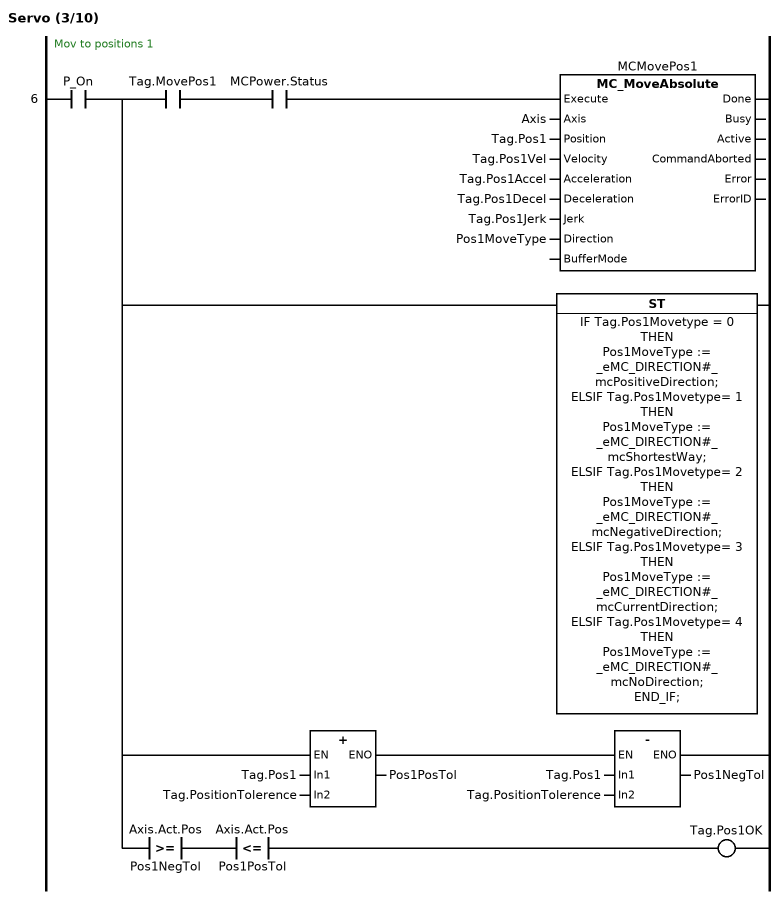
(* [picture p96: Servo, rungs 6-6] *)
(* Rung 6: Mov to positions 1 *)
MCMovePos1(Execute := P_On AND Tag.MovePos1 AND MCPower.Status, Axis := Axis, Position := Tag.Pos1, Velocity := Tag.Pos1Vel, Acceleration := Tag.Pos1Accel, Deceleration := Tag.Pos1Decel, Jerk := Tag.Pos1Jerk, Direction := Pos1MoveType);
IF P_On THEN
    IF Tag.Pos1Movetype = 0 THEN
    Pos1MoveType := _eMC_DIRECTION#_mcPositiveDirection;
    ELSIF Tag.Pos1Movetype= 1 THEN
    Pos1MoveType := _eMC_DIRECTION#_mcShortestWay;
    ELSIF Tag.Pos1Movetype= 2 THEN
    Pos1MoveType := _eMC_DIRECTION#_mcNegativeDirection;
    ELSIF Tag.Pos1Movetype= 3 THEN
    Pos1MoveType := _eMC_DIRECTION#_mcCurrentDirection;
    ELSIF Tag.Pos1Movetype= 4 THEN
    Pos1MoveType := _eMC_DIRECTION#_mcNoDirection;
    END_IF;
END_IF;
IF P_On THEN
    Pos1PosTol := Tag.Pos1 + Tag.PositionTolerence;
    Pos1NegTol := Tag.Pos1 - Tag.PositionTolerence;
END_IF;
Tag.Pos1OK := P_On AND (Axis.Act.Pos >= Pos1NegTol) AND (Axis.Act.Pos <= Pos1PosTol);

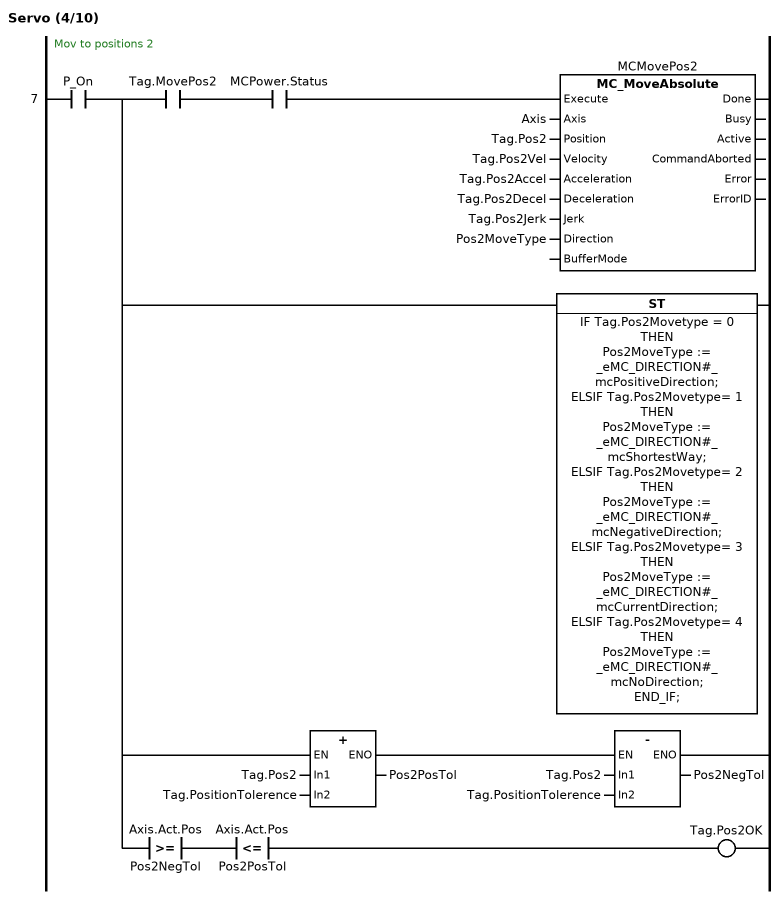
(* Rung 7: Mov to positions 2 *)
MCMovePos2(Execute := P_On AND Tag.MovePos2 AND MCPower.Status, Axis := Axis, Position := Tag.Pos2, Velocity := Tag.Pos2Vel, Acceleration := Tag.Pos2Accel, Deceleration := Tag.Pos2Decel, Jerk := Tag.Pos2Jerk, Direction := Pos2MoveType);
IF P_On THEN
    IF Tag.Pos2Movetype = 0 THEN
    Pos2MoveType := _eMC_DIRECTION#_mcPositiveDirection;
    ELSIF Tag.Pos2Movetype= 1 THEN
    Pos2MoveType := _eMC_DIRECTION#_mcShortestWay;
    ELSIF Tag.Pos2Movetype= 2 THEN
    Pos2MoveType := _eMC_DIRECTION#_mcNegativeDirection;
    ELSIF Tag.Pos2Movetype= 3 THEN
    Pos2MoveType := _eMC_DIRECTION#_mcCurrentDirection;
    ELSIF Tag.Pos2Movetype= 4 THEN
    Pos2MoveType := _eMC_DIRECTION#_mcNoDirection;
    END_IF;
END_IF;
IF P_On THEN
    Pos2PosTol := Tag.Pos2 + Tag.PositionTolerence;
    Pos2NegTol := Tag.Pos2 - Tag.PositionTolerence;
END_IF;
Tag.Pos2OK := P_On AND (Axis.Act.Pos >= Pos2NegTol) AND (Axis.Act.Pos <= Pos2PosTol);

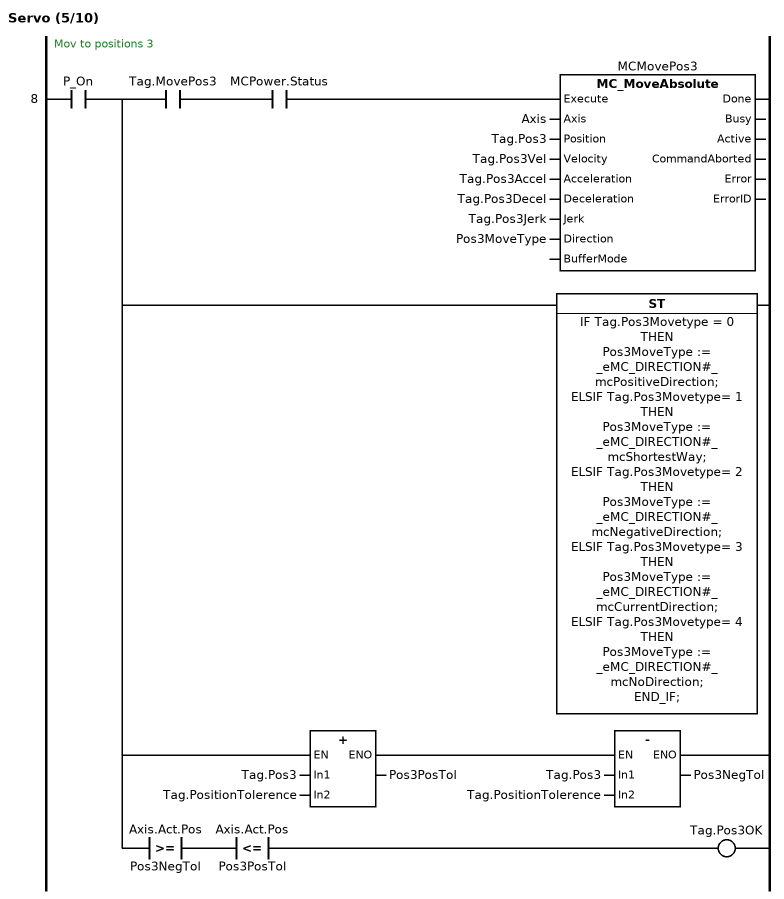
(* Rung 8: Mov to positions 3 *)
MCMovePos3(Execute := P_On AND Tag.MovePos3 AND MCPower.Status, Axis := Axis, Position := Tag.Pos3, Velocity := Tag.Pos3Vel, Acceleration := Tag.Pos3Accel, Deceleration := Tag.Pos3Decel, Jerk := Tag.Pos3Jerk, Direction := Pos3MoveType);
IF P_On THEN
    IF Tag.Pos3Movetype = 0 THEN
    Pos3MoveType := _eMC_DIRECTION#_mcPositiveDirection;
    ELSIF Tag.Pos3Movetype= 1 THEN
    Pos3MoveType := _eMC_DIRECTION#_mcShortestWay;
    ELSIF Tag.Pos3Movetype= 2 THEN
    Pos3MoveType := _eMC_DIRECTION#_mcNegativeDirection;
    ELSIF Tag.Pos3Movetype= 3 THEN
    Pos3MoveType := _eMC_DIRECTION#_mcCurrentDirection;
    ELSIF Tag.Pos3Movetype= 4 THEN
    Pos3MoveType := _eMC_DIRECTION#_mcNoDirection;
    END_IF;
END_IF;
IF P_On THEN
    Pos3PosTol := Tag.Pos3 + Tag.PositionTolerence;
    Pos3NegTol := Tag.Pos3 - Tag.PositionTolerence;
END_IF;
Tag.Pos3OK := P_On AND (Axis.Act.Pos >= Pos3NegTol) AND (Axis.Act.Pos <= Pos3PosTol);

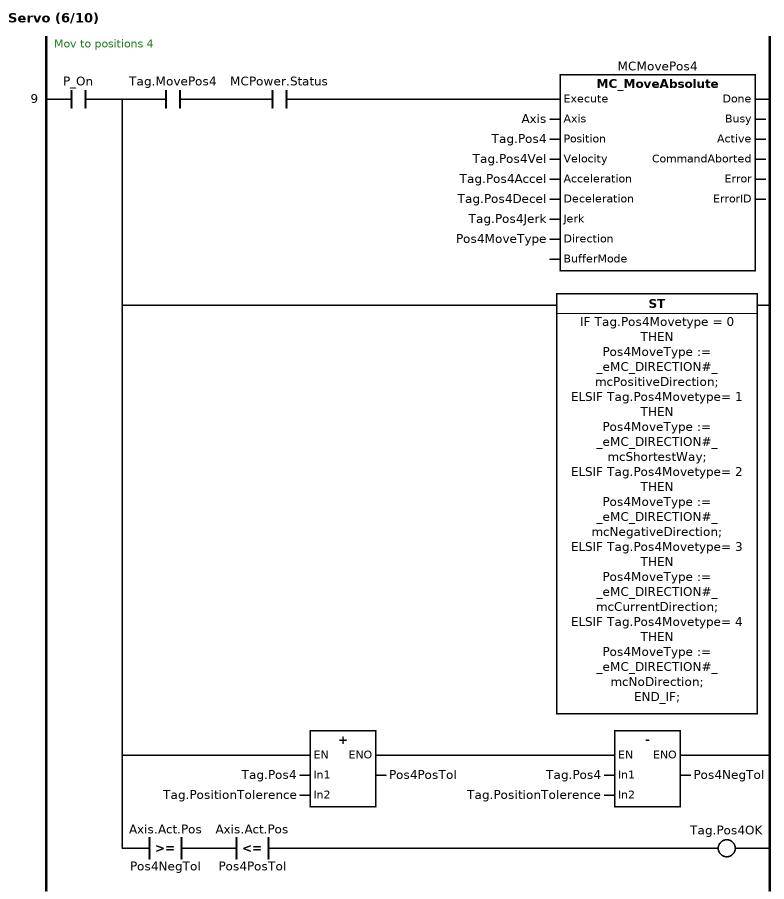
(* Rung 9: Mov to positions 4 *)
MCMovePos4(Execute := P_On AND Tag.MovePos4 AND MCPower.Status, Axis := Axis, Position := Tag.Pos4, Velocity := Tag.Pos4Vel, Acceleration := Tag.Pos4Accel, Deceleration := Tag.Pos4Decel, Jerk := Tag.Pos4Jerk, Direction := Pos4MoveType);
IF P_On THEN
    IF Tag.Pos4Movetype = 0 THEN
    Pos4MoveType := _eMC_DIRECTION#_mcPositiveDirection;
    ELSIF Tag.Pos4Movetype= 1 THEN
    Pos4MoveType := _eMC_DIRECTION#_mcShortestWay;
    ELSIF Tag.Pos4Movetype= 2 THEN
    Pos4MoveType := _eMC_DIRECTION#_mcNegativeDirection;
    ELSIF Tag.Pos4Movetype= 3 THEN
    Pos4MoveType := _eMC_DIRECTION#_mcCurrentDirection;
    ELSIF Tag.Pos4Movetype= 4 THEN
    Pos4MoveType := _eMC_DIRECTION#_mcNoDirection;
    END_IF;
END_IF;
IF P_On THEN
    Pos4PosTol := Tag.Pos4 + Tag.PositionTolerence;
    Pos4NegTol := Tag.Pos4 - Tag.PositionTolerence;
END_IF;
Tag.Pos4OK := P_On AND (Axis.Act.Pos >= Pos4NegTol) AND (Axis.Act.Pos <= Pos4PosTol);

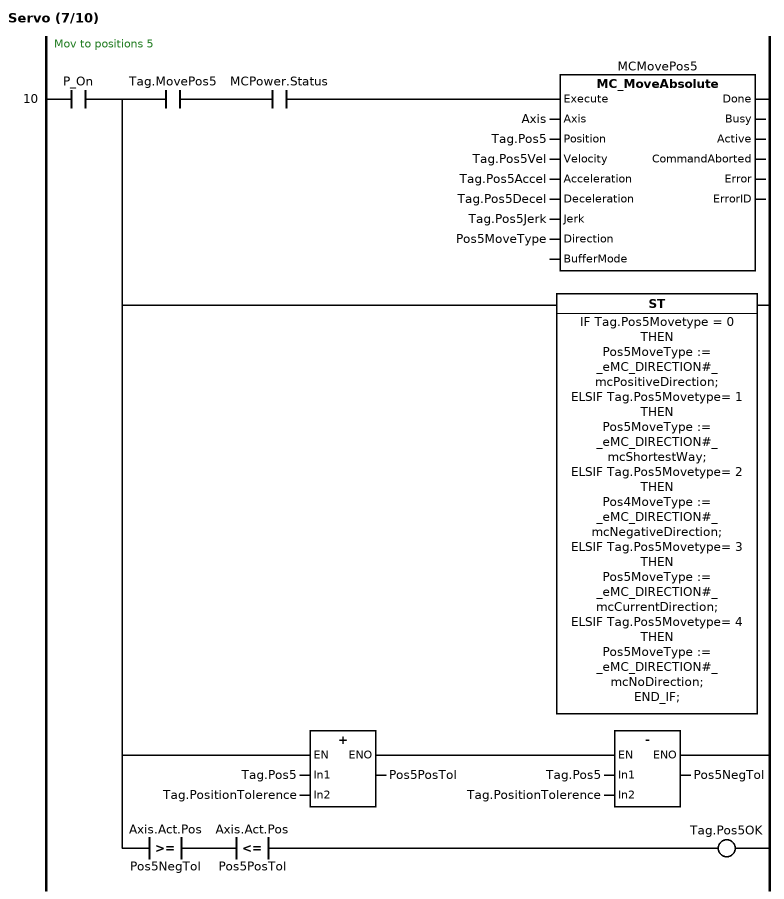
(* Rung 10: Mov to positions 5 *)
MCMovePos5(Execute := P_On AND Tag.MovePos5 AND MCPower.Status, Axis := Axis, Position := Tag.Pos5, Velocity := Tag.Pos5Vel, Acceleration := Tag.Pos5Accel, Deceleration := Tag.Pos5Decel, Jerk := Tag.Pos5Jerk, Direction := Pos5MoveType);
IF P_On THEN
    IF Tag.Pos5Movetype = 0 THEN
    Pos5MoveType := _eMC_DIRECTION#_mcPositiveDirection;
    ELSIF Tag.Pos5Movetype= 1 THEN
    Pos5MoveType := _eMC_DIRECTION#_mcShortestWay;
    ELSIF Tag.Pos5Movetype= 2 THEN
    Pos4MoveType := _eMC_DIRECTION#_mcNegativeDirection;
    ELSIF Tag.Pos5Movetype= 3 THEN
    Pos5MoveType := _eMC_DIRECTION#_mcCurrentDirection;
    ELSIF Tag.Pos5Movetype= 4 THEN
    Pos5MoveType := _eMC_DIRECTION#_mcNoDirection;
    END_IF;
END_IF;
IF P_On THEN
    Pos5PosTol := Tag.Pos5 + Tag.PositionTolerence;
    Pos5NegTol := Tag.Pos5 - Tag.PositionTolerence;
END_IF;
Tag.Pos5OK := P_On AND (Axis.Act.Pos >= Pos5NegTol) AND (Axis.Act.Pos <= Pos5PosTol);

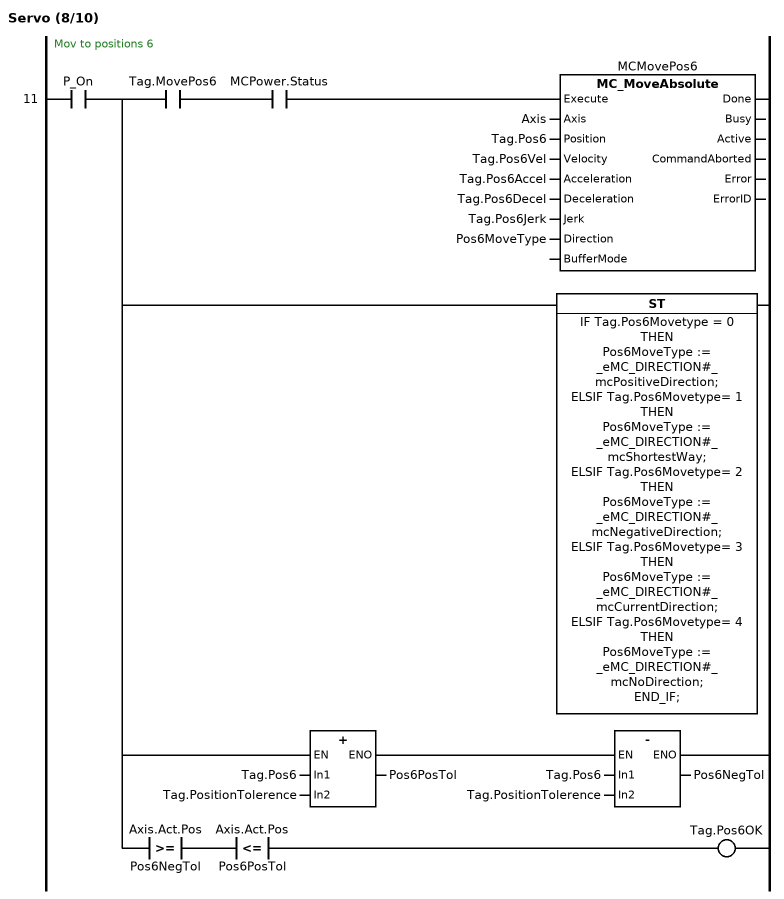
(* Rung 11: Mov to positions 6 *)
MCMovePos6(Execute := P_On AND Tag.MovePos6 AND MCPower.Status, Axis := Axis, Position := Tag.Pos6, Velocity := Tag.Pos6Vel, Acceleration := Tag.Pos6Accel, Deceleration := Tag.Pos6Decel, Jerk := Tag.Pos6Jerk, Direction := Pos6MoveType);
IF P_On THEN
    IF Tag.Pos6Movetype = 0 THEN
    Pos6MoveType := _eMC_DIRECTION#_mcPositiveDirection;
    ELSIF Tag.Pos6Movetype= 1 THEN
    Pos6MoveType := _eMC_DIRECTION#_mcShortestWay;
    ELSIF Tag.Pos6Movetype= 2 THEN
    Pos6MoveType := _eMC_DIRECTION#_mcNegativeDirection;
    ELSIF Tag.Pos6Movetype= 3 THEN
    Pos6MoveType := _eMC_DIRECTION#_mcCurrentDirection;
    ELSIF Tag.Pos6Movetype= 4 THEN
    Pos6MoveType := _eMC_DIRECTION#_mcNoDirection;
    END_IF;
END_IF;
IF P_On THEN
    Pos6PosTol := Tag.Pos6 + Tag.PositionTolerence;
    Pos6NegTol := Tag.Pos6 - Tag.PositionTolerence;
END_IF;
Tag.Pos6OK := P_On AND (Axis.Act.Pos >= Pos6NegTol) AND (Axis.Act.Pos <= Pos6PosTol);

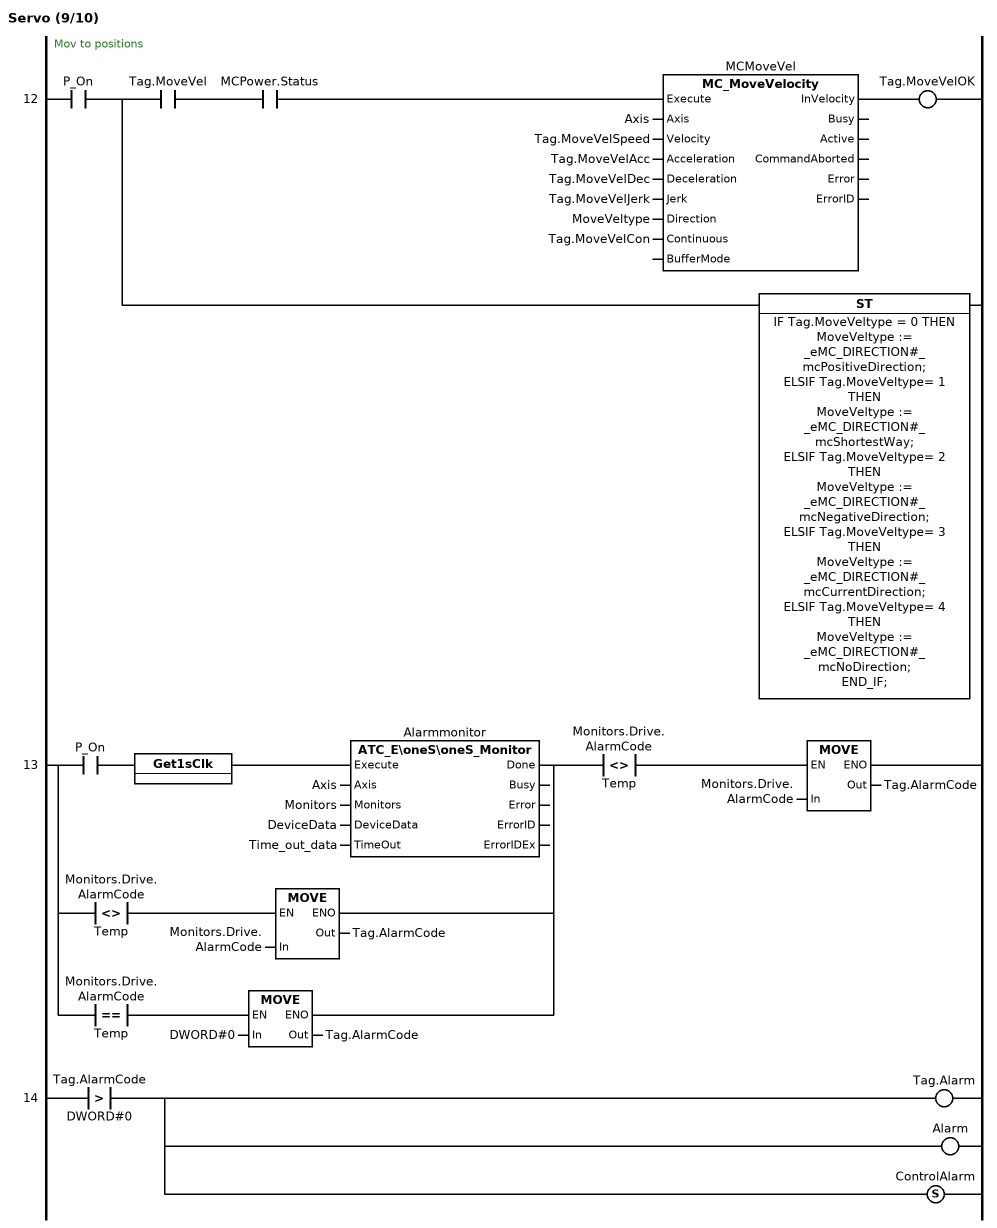
(* Rung 12: Mov to positions *)
MCMoveVel(Execute := P_On AND Tag.MoveVel AND MCPower.Status, Axis := Axis, Velocity := Tag.MoveVelSpeed, Acceleration := Tag.MoveVelAcc, Deceleration := Tag.MoveVelDec, Jerk := Tag.MoveVelJerk, Direction := MoveVeltype, Continuous := Tag.MoveVelCon);
Tag.MoveVelOK := MCMoveVel.InVelocity;
IF P_On THEN
    IF Tag.MoveVeltype = 0 THEN
    MoveVeltype := _eMC_DIRECTION#_mcPositiveDirection;
    ELSIF Tag.MoveVeltype= 1 THEN
    MoveVeltype := _eMC_DIRECTION#_mcShortestWay;
    ELSIF Tag.MoveVeltype= 2 THEN
    MoveVeltype := _eMC_DIRECTION#_mcNegativeDirection;
    ELSIF Tag.MoveVeltype= 3 THEN
    MoveVeltype := _eMC_DIRECTION#_mcCurrentDirection;
    ELSIF Tag.MoveVeltype= 4 THEN
    MoveVeltype := _eMC_DIRECTION#_mcNoDirection;
    END_IF;
END_IF;
(* Rung 13 *)
Alarmmonitor(Execute := P_On AND Get1sClk(), Axis := Axis, Monitors := Monitors, DeviceData := DeviceData, TimeOut := Time_out_data);
IF Monitors.Drive.AlarmCode <> Temp THEN Tag.AlarmCode := Monitors.Drive.AlarmCode; END_IF;
IF Monitors.Drive.AlarmCode = Temp THEN Tag.AlarmCode := DWORD#0; END_IF;
IF (Alarmmonitor.Done OR (Monitors.Drive.AlarmCode <> Temp) OR (Monitors.Drive.AlarmCode = Temp)) AND (Monitors.Drive.AlarmCode <> Temp) THEN
    Tag.AlarmCode := Monitors.Drive.AlarmCode;
END_IF;
(* Rung 14 *)
_p1 := Tag.AlarmCode > DWORD#0;
Tag.Alarm := _p1;
Alarm := _p1;
IF _p1 THEN ControlAlarm := TRUE; END_IF;

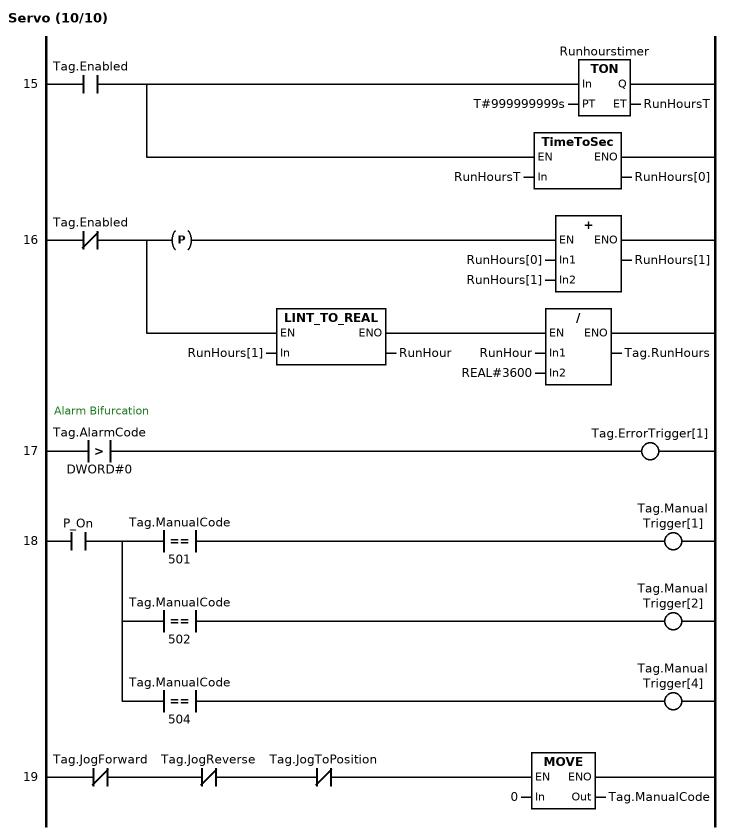
(* Rung 15 *)
Runhourstimer(In := Tag.Enabled, PT := T#999999999s, ET => RunHoursT);
IF Tag.Enabled THEN RunHours[0] := TimeToSec(In := RunHoursT); END_IF;
(* Rung 16 *)
_e2(CLK := NOT Tag.Enabled);
IF _e2.Q THEN RunHours[1] := RunHours[0] + RunHours[1]; END_IF;
IF NOT Tag.Enabled THEN
    RunHour := LINT_TO_REAL(In := RunHours[1]);
    Tag.RunHours := RunHour / REAL#3600;
END_IF;
(* Rung 17: Alarm Bifurcation *)
Tag.ErrorTrigger[1] := Tag.AlarmCode > DWORD#0;
(* Rung 18 *)
Tag.ManualTrigger[1] := P_On AND (Tag.ManualCode = 501);
Tag.ManualTrigger[2] := P_On AND (Tag.ManualCode = 502);
Tag.ManualTrigger[4] := P_On AND (Tag.ManualCode = 504);
(* Rung 19 *)
IF NOT Tag.JogForward AND NOT Tag.JogReverse AND NOT Tag.JogToPosition THEN Tag.ManualCode := 0; END_IF;
END_FUNCTION_BLOCK

FUNCTION_BLOCK MiscIN
VAR
    Powerup : BOOL;
    IN : BOOL;
    DebounceON : TON;
    Debounceoff : TON;
    In_Fault_Timer : TON;
    Timecal1 : LREAL;
    Timecal2 : LINT;
    DebounceONtime : TIME;
    Timecal3 : LINT;
    Timecal4 : LREAL;
    AccumulatedON : TIME;
    Timecal5 : LREAL;
    Timecal6 : LINT;
    DebounceOFFtime : TIME;
    Timecal7 : LINT;
    Timecal8 : LREAL;
    AccumulatedOFF : TIME;
    Timecal9 : LREAL;
    Timecal10 : LINT;
    Input_Fault_Time : TIME;
    Timecal11 : LINT;
    Timecal12 : LREAL;
    Input_Fault_Time_Acc : TIME;
END_VAR
VAR_OUTPUT
    EnableOut : BOOL;
END_VAR
VAR_INPUT
    input : BOOL;
    Accnowledge : BOOL;
END_VAR
VAR_IN_OUT
    tag : MiscInD;
END_VAR
VAR_OUTPUT
    Alarm : BOOL;
END_VAR
VAR_IN_OUT
    ControlAlarm : BOOL;
END_VAR
VAR
    _p1 : BOOL;
    _p2 : BOOL;
    _p3 : BOOL;
    _p4 : BOOL;
    _p5 : BOOL;
END_VAR
(* ladder, written here as Structured Text *)

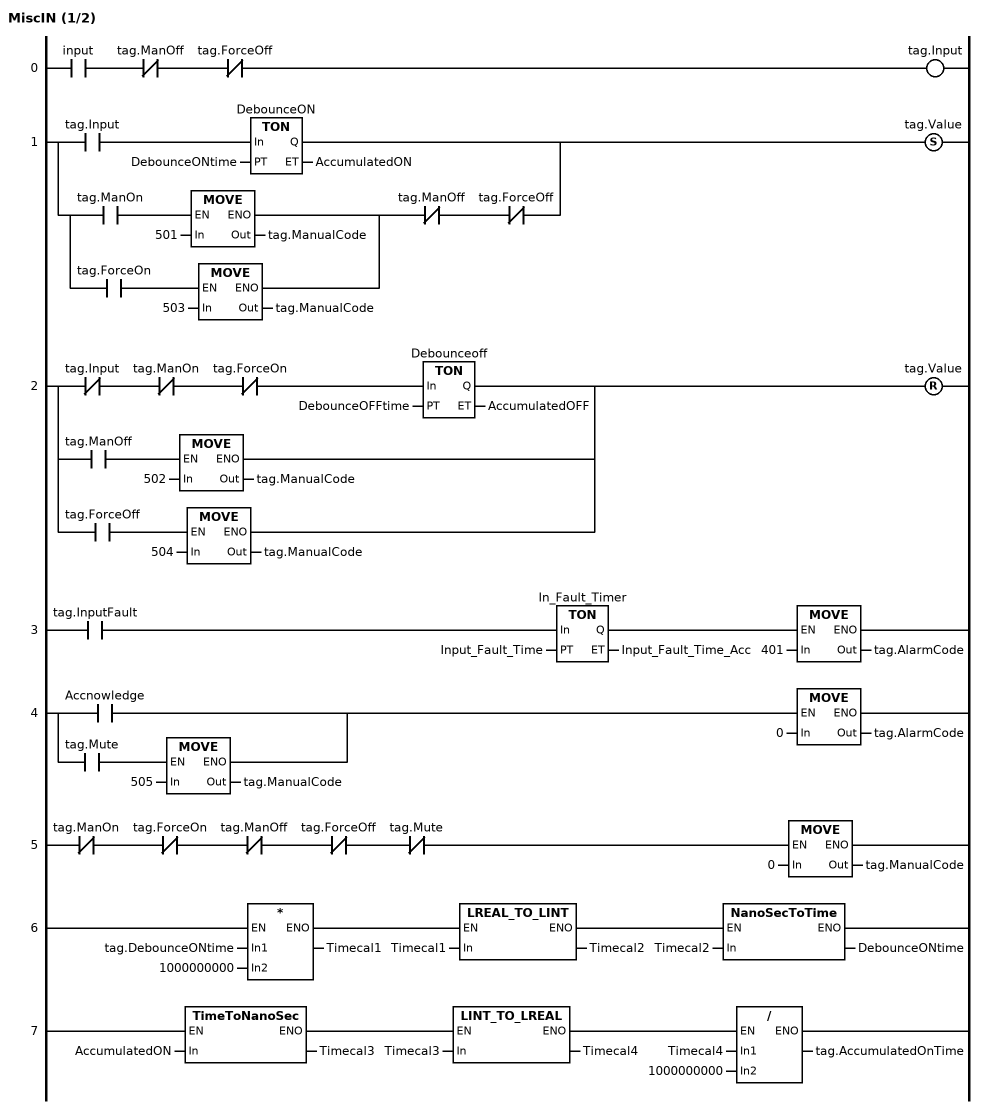
(* Rung 0 *)
tag.Input := input AND NOT tag.ManOff AND NOT tag.ForceOff;
(* Rung 1 *)
DebounceON(In := tag.Input, PT := DebounceONtime, ET => AccumulatedON);
_p1 := tag.ManOn;
IF _p1 THEN tag.ManualCode := 501; END_IF;
_p2 := tag.ForceOn;
IF _p2 THEN tag.ManualCode := 503; END_IF;
IF DebounceON.Q OR ((_p1 OR _p2) AND NOT tag.ManOff AND NOT tag.ForceOff) THEN tag.Value := TRUE; END_IF;
(* Rung 2 *)
Debounceoff(In := NOT tag.Input AND NOT tag.ManOn AND NOT tag.ForceOn, PT := DebounceOFFtime, ET => AccumulatedOFF);
_p3 := tag.ManOff;
IF _p3 THEN tag.ManualCode := 502; END_IF;
_p4 := tag.ForceOff;
IF _p4 THEN tag.ManualCode := 504; END_IF;
IF Debounceoff.Q OR _p3 OR _p4 THEN tag.Value := FALSE; END_IF;
(* Rung 3 *)
In_Fault_Timer(In := tag.InputFault, PT := Input_Fault_Time, ET => Input_Fault_Time_Acc);
IF In_Fault_Timer.Q THEN tag.AlarmCode := 401; END_IF;
(* Rung 4 *)
_p5 := tag.Mute;
IF _p5 THEN tag.ManualCode := 505; END_IF;
IF Accnowledge OR _p5 THEN tag.AlarmCode := 0; END_IF;
(* Rung 5 *)
IF NOT tag.ManOn AND NOT tag.ForceOn AND NOT tag.ManOff AND NOT tag.ForceOff AND NOT tag.Mute THEN
    tag.ManualCode := 0;
END_IF;
(* Rung 6 *)
Timecal1 := tag.DebounceONtime * 1000000000;
Timecal2 := LREAL_TO_LINT(In := Timecal1);
DebounceONtime := NanoSecToTime(In := Timecal2);
(* Rung 7 *)
Timecal3 := TimeToNanoSec(In := AccumulatedON);
Timecal4 := LINT_TO_LREAL(In := Timecal3);
tag.AccumulatedOnTime := Timecal4 / 1000000000;

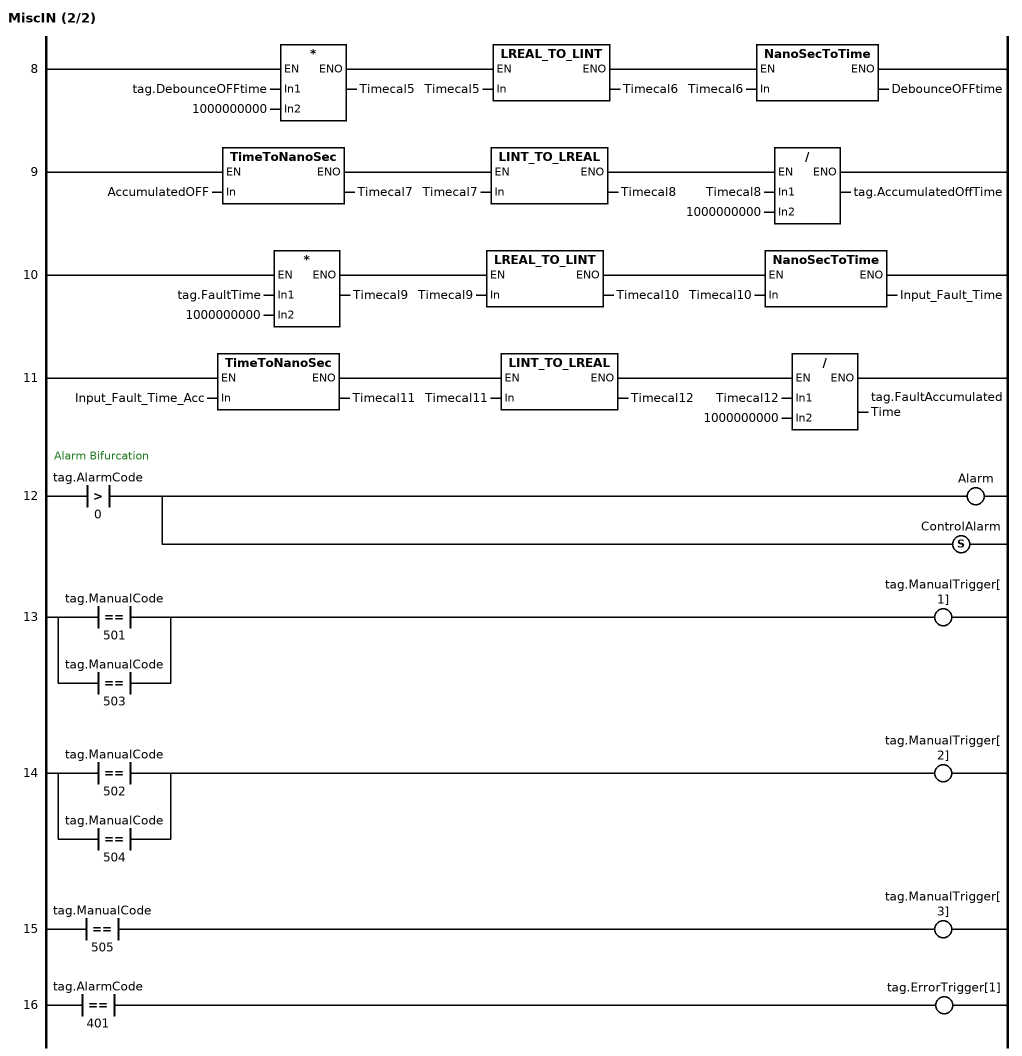
(* Rung 8 *)
Timecal5 := tag.DebounceOFFtime * 1000000000;
Timecal6 := LREAL_TO_LINT(In := Timecal5);
DebounceOFFtime := NanoSecToTime(In := Timecal6);
(* Rung 9 *)
Timecal7 := TimeToNanoSec(In := AccumulatedOFF);
Timecal8 := LINT_TO_LREAL(In := Timecal7);
tag.AccumulatedOffTime := Timecal8 / 1000000000;
(* Rung 10 *)
Timecal9 := tag.FaultTime * 1000000000;
Timecal10 := LREAL_TO_LINT(In := Timecal9);
Input_Fault_Time := NanoSecToTime(In := Timecal10);
(* Rung 11 *)
Timecal11 := TimeToNanoSec(In := Input_Fault_Time_Acc);
Timecal12 := LINT_TO_LREAL(In := Timecal11);
tag.FaultAccumulatedTime := Timecal12 / 1000000000;
(* Rung 12: Alarm Bifurcation *)
Alarm := tag.AlarmCode > 0;
IF tag.AlarmCode > 0 THEN ControlAlarm := TRUE; END_IF;
(* Rung 13 *)
tag.ManualTrigger[1] := (tag.ManualCode = 501) OR (tag.ManualCode = 503);
(* Rung 14 *)
tag.ManualTrigger[2] := (tag.ManualCode = 502) OR (tag.ManualCode = 504);
(* Rung 15 *)
tag.ManualTrigger[3] := tag.ManualCode = 505;
(* Rung 16 *)
tag.ErrorTrigger[1] := tag.AlarmCode = 401;
END_FUNCTION_BLOCK

FUNCTION_BLOCK Motor
VAR
    Forward : BOOL;
    Reverse : BOOL;
    FeedBackOffTimer : TON;
END_VAR
VAR RETAIN
    Faulttime : TIME;
END_VAR
VAR
    MotorFault : BOOL;
    FeedBackOnTimer : TON;
    Faulttime1Acc : TIME;
    MotorFaultRev : BOOL;
    Timecal7 : LREAL;
    Timecal8 : LINT;
    Timecal9 : LINT;
    Timecal10 : LREAL;
    FaulttimeAcc : TIME;
    RunHoursT : TIME;
    RunHours : ARRAY[0..1] OF LINT;
    RunHour : REAL;
    RunHoursTimer : TON;
    MotorFaultoff : BOOL;
    FeedBackOffTimer1 : TON;
END_VAR
VAR_INPUT
    Enable : BOOL;
END_VAR
VAR_OUTPUT
    Enableout : BOOL;
    OutputForward : BOOL;
    OutputReverse : BOOL;
END_VAR
VAR_INPUT
    RunFeedBack : BOOL;
END_VAR
VAR_IN_OUT
    Tag : MotorD;
END_VAR
VAR_OUTPUT
    Alarm : BOOL;
END_VAR
VAR_IN_OUT
    ControlCom : System;
END_VAR
VAR
    _e1 : R_TRIG;
    _e2 : R_TRIG;
    _p3 : BOOL;
    _e4 : R_TRIG;
    _e5 : R_TRIG;
    _p6 : BOOL;
    _p7 : BOOL;
    _p8 : BOOL;
    _p9 : BOOL;
    _e10 : R_TRIG;
    _e11 : R_TRIG;
    _p12 : BOOL;
END_VAR
(* ladder, written here as Structured Text *)

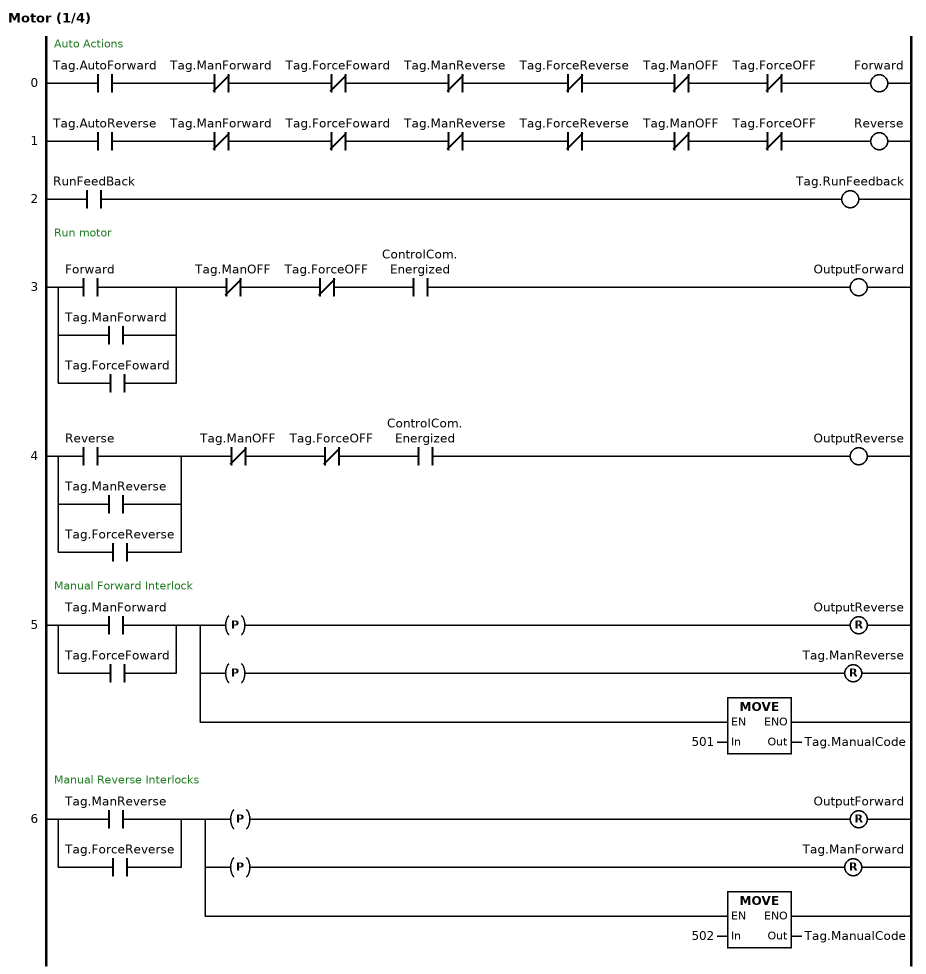
(* Rung 0: Auto Actions *)
Forward := Tag.AutoForward AND NOT Tag.ManForward AND NOT Tag.ForceFoward AND NOT Tag.ManReverse AND NOT Tag.ForceReverse AND NOT Tag.ManOFF AND NOT Tag.ForceOFF;
(* Rung 1 *)
Reverse := Tag.AutoReverse AND NOT Tag.ManForward AND NOT Tag.ForceFoward AND NOT Tag.ManReverse AND NOT Tag.ForceReverse AND NOT Tag.ManOFF AND NOT Tag.ForceOFF;
(* Rung 2 *)
Tag.RunFeedback := RunFeedBack;
(* Rung 3: Run motor *)
OutputForward := (Forward OR Tag.ManForward OR Tag.ForceFoward) AND NOT Tag.ManOFF AND NOT Tag.ForceOFF AND ControlCom.Energized;
(* Rung 4 *)
OutputReverse := (Reverse OR Tag.ManReverse OR Tag.ForceReverse) AND NOT Tag.ManOFF AND NOT Tag.ForceOFF AND ControlCom.Energized;
(* Rung 5: Manual Forward Interlock *)
_e1(CLK := Tag.ManForward OR Tag.ForceFoward);
IF _e1.Q THEN OutputReverse := FALSE; END_IF;
_e2(CLK := Tag.ManForward OR Tag.ForceFoward);
_p3 := Tag.ManForward OR Tag.ForceFoward;
IF _e2.Q THEN Tag.ManReverse := FALSE; END_IF;
IF _p3 THEN Tag.ManualCode := 501; END_IF;
(* Rung 6: Manual Reverse Interlocks *)
_e4(CLK := Tag.ManReverse OR Tag.ForceReverse);
IF _e4.Q THEN OutputForward := FALSE; END_IF;
_e5(CLK := Tag.ManReverse OR Tag.ForceReverse);
_p6 := Tag.ManReverse OR Tag.ForceReverse;
IF _e5.Q THEN Tag.ManForward := FALSE; END_IF;
IF _p6 THEN Tag.ManualCode := 502; END_IF;

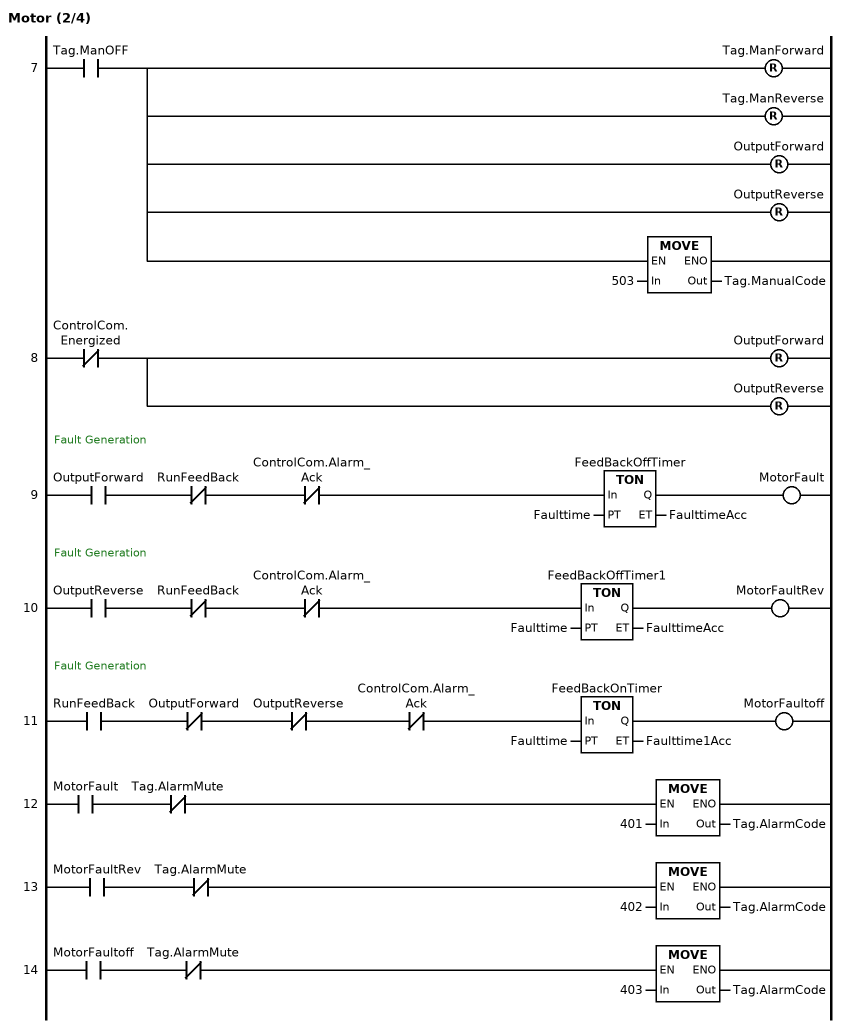
(* Rung 7 *)
_p7 := Tag.ManOFF;
IF _p7 THEN
    Tag.ManForward := FALSE;
    Tag.ManReverse := FALSE;
    OutputForward := FALSE;
    OutputReverse := FALSE;
    Tag.ManualCode := 503;
END_IF;
(* Rung 8 *)
IF NOT ControlCom.Energized THEN
    OutputForward := FALSE;
    OutputReverse := FALSE;
END_IF;
(* Rung 9: Fault Generation *)
FeedBackOffTimer(In := OutputForward AND NOT RunFeedBack AND NOT ControlCom.Alarm_Ack, PT := Faulttime, ET => FaulttimeAcc);
MotorFault := FeedBackOffTimer.Q;
(* Rung 10: Fault Generation *)
FeedBackOffTimer1(In := OutputReverse AND NOT RunFeedBack AND NOT ControlCom.Alarm_Ack, PT := Faulttime, ET => FaulttimeAcc);
MotorFaultRev := FeedBackOffTimer1.Q;
(* Rung 11: Fault Generation *)
FeedBackOnTimer(In := RunFeedBack AND NOT OutputForward AND NOT OutputReverse AND NOT ControlCom.Alarm_Ack, PT := Faulttime, ET => Faulttime1Acc);
MotorFaultoff := FeedBackOnTimer.Q;
(* Rung 12 *)
IF MotorFault AND NOT Tag.AlarmMute THEN Tag.AlarmCode := 401; END_IF;
(* Rung 13 *)
IF MotorFaultRev AND NOT Tag.AlarmMute THEN Tag.AlarmCode := 402; END_IF;
(* Rung 14 *)
IF MotorFaultoff AND NOT Tag.AlarmMute THEN Tag.AlarmCode := 403; END_IF;

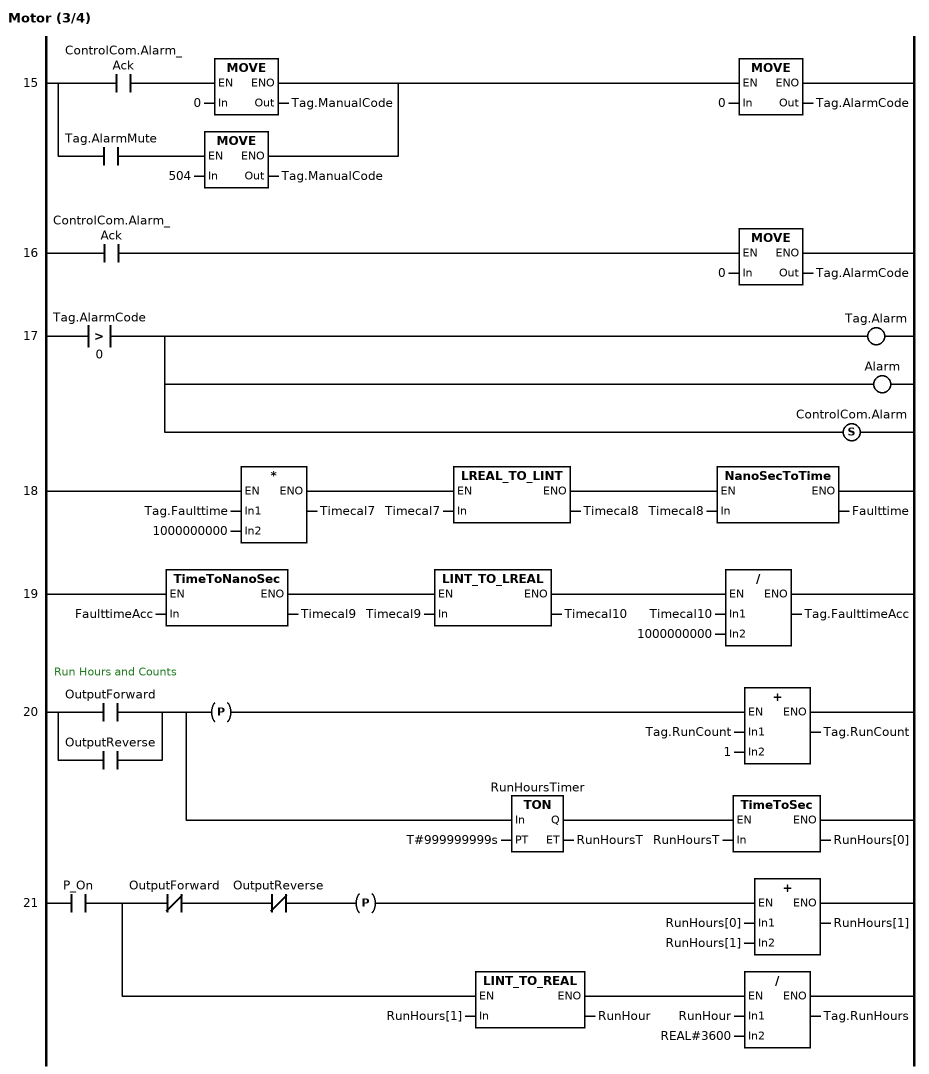
(* Rung 15 *)
IF ControlCom.Alarm_Ack THEN Tag.ManualCode := 0; END_IF;
_p8 := Tag.AlarmMute;
IF _p8 THEN Tag.ManualCode := 504; END_IF;
IF ControlCom.Alarm_Ack OR _p8 THEN Tag.AlarmCode := 0; END_IF;
(* Rung 16 *)
IF ControlCom.Alarm_Ack THEN Tag.AlarmCode := 0; END_IF;
(* Rung 17 *)
_p9 := Tag.AlarmCode > 0;
Tag.Alarm := _p9;
Alarm := _p9;
IF _p9 THEN ControlCom.Alarm := TRUE; END_IF;
(* Rung 18 *)
Timecal7 := Tag.Faulttime * 1000000000;
Timecal8 := LREAL_TO_LINT(In := Timecal7);
Faulttime := NanoSecToTime(In := Timecal8);
(* Rung 19 *)
Timecal9 := TimeToNanoSec(In := FaulttimeAcc);
Timecal10 := LINT_TO_LREAL(In := Timecal9);
Tag.FaulttimeAcc := Timecal10 / 1000000000;
(* Rung 20: Run Hours and Counts *)
_e10(CLK := OutputForward OR OutputReverse);
IF _e10.Q THEN Tag.RunCount := Tag.RunCount + 1; END_IF;
RunHoursTimer(In := OutputForward OR OutputReverse, PT := T#999999999s, ET => RunHoursT);
IF RunHoursTimer.Q THEN RunHours[0] := TimeToSec(In := RunHoursT); END_IF;
(* Rung 21 *)
_e11(CLK := P_On AND NOT OutputForward AND NOT OutputReverse);
IF _e11.Q THEN RunHours[1] := RunHours[0] + RunHours[1]; END_IF;
IF P_On THEN
    RunHour := LINT_TO_REAL(In := RunHours[1]);
    Tag.RunHours := RunHour / REAL#3600;
END_IF;

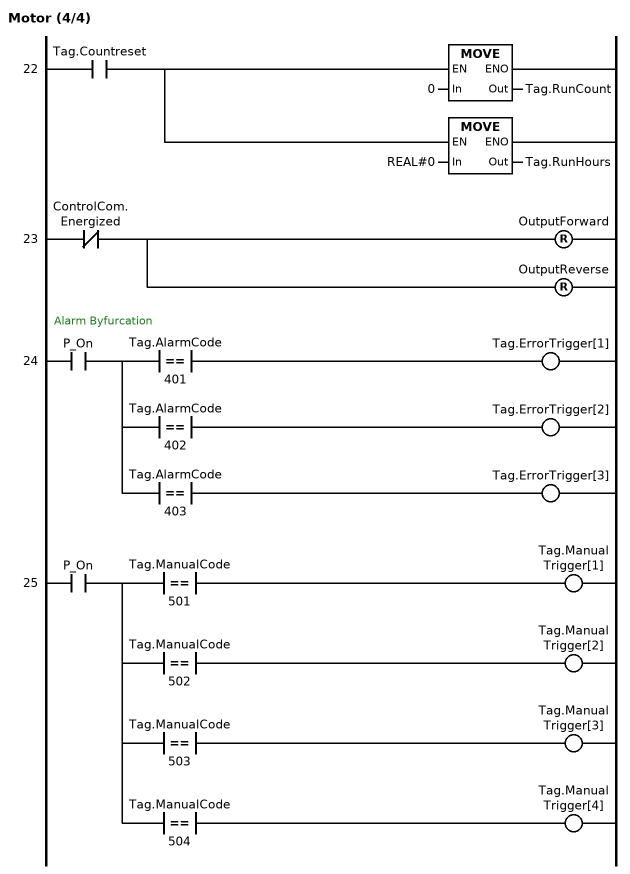
(* Rung 22 *)
_p12 := Tag.Countreset;
IF _p12 THEN
    Tag.RunCount := 0;
    Tag.RunHours := REAL#0;
END_IF;
(* Rung 23 *)
IF NOT ControlCom.Energized THEN
    OutputForward := FALSE;
    OutputReverse := FALSE;
END_IF;
(* Rung 24: Alarm Byfurcation *)
Tag.ErrorTrigger[1] := P_On AND (Tag.AlarmCode = 401);
Tag.ErrorTrigger[2] := P_On AND (Tag.AlarmCode = 402);
Tag.ErrorTrigger[3] := P_On AND (Tag.AlarmCode = 403);
(* Rung 25 *)
Tag.ManualTrigger[1] := P_On AND (Tag.ManualCode = 501);
Tag.ManualTrigger[2] := P_On AND (Tag.ManualCode = 502);
Tag.ManualTrigger[3] := P_On AND (Tag.ManualCode = 503);
Tag.ManualTrigger[4] := P_On AND (Tag.ManualCode = 504);
END_FUNCTION_BLOCK

FUNCTION_BLOCK MotorVSD
VAR
    Forward : BOOL;
    Reverse : BOOL;
    FeedBackOffTimer : TON;
END_VAR
VAR RETAIN
    Faulttime : TIME;
END_VAR
VAR
    MotorFault : BOOL;
    FeedBackOnTimer : TON;
    Faulttime1Acc : TIME;
    MotorFaultRev : BOOL;
    Timecal7 : LREAL;
    Timecal8 : LINT;
    Timecal9 : LINT;
    Timecal10 : LREAL;
    FaulttimeAcc : TIME;
    OutputForward : BOOL;
    OutputReverse : BOOL;
    MotorFaultFor : BOOL;
    FeedBackOffTimerFor : TON;
    FeedBackOnTimerRev : TON;
    Faulttime2Acc : TIME;
    RunHoursTimer : TON;
    RunHoursT : TIME;
    RunHours : ARRAY[0..1] OF LINT;
    RunHour : REAL;
END_VAR
VAR_INPUT
    Enable : BOOL;
END_VAR
VAR_OUTPUT
    Enableout : BOOL;
END_VAR
VAR_IN_OUT
    Tag : MotorVSDD;
END_VAR
VAR_OUTPUT
    DirectionOut : WORD;
    SpeedOut : UINT;
END_VAR
VAR_INPUT
    RunFeedBack : WORD;
END_VAR
VAR_OUTPUT
    Alarm : BOOL;
END_VAR
VAR_IN_OUT
    ControlCom : System;
END_VAR
VAR_EXTERNAL
    Zcomm : ARRAY[0..31] OF BOOL;
END_VAR
VAR
    _p1 : BOOL;
    _e2 : R_TRIG;
    _e3 : R_TRIG;
    _p4 : BOOL;
    _e5 : R_TRIG;
    _e6 : R_TRIG;
    _p7 : BOOL;
    _p8 : BOOL;
    _p9 : BOOL;
    _e10 : R_TRIG;
    _e11 : R_TRIG;
    _p12 : BOOL;
END_VAR
(* ladder, written here as Structured Text *)

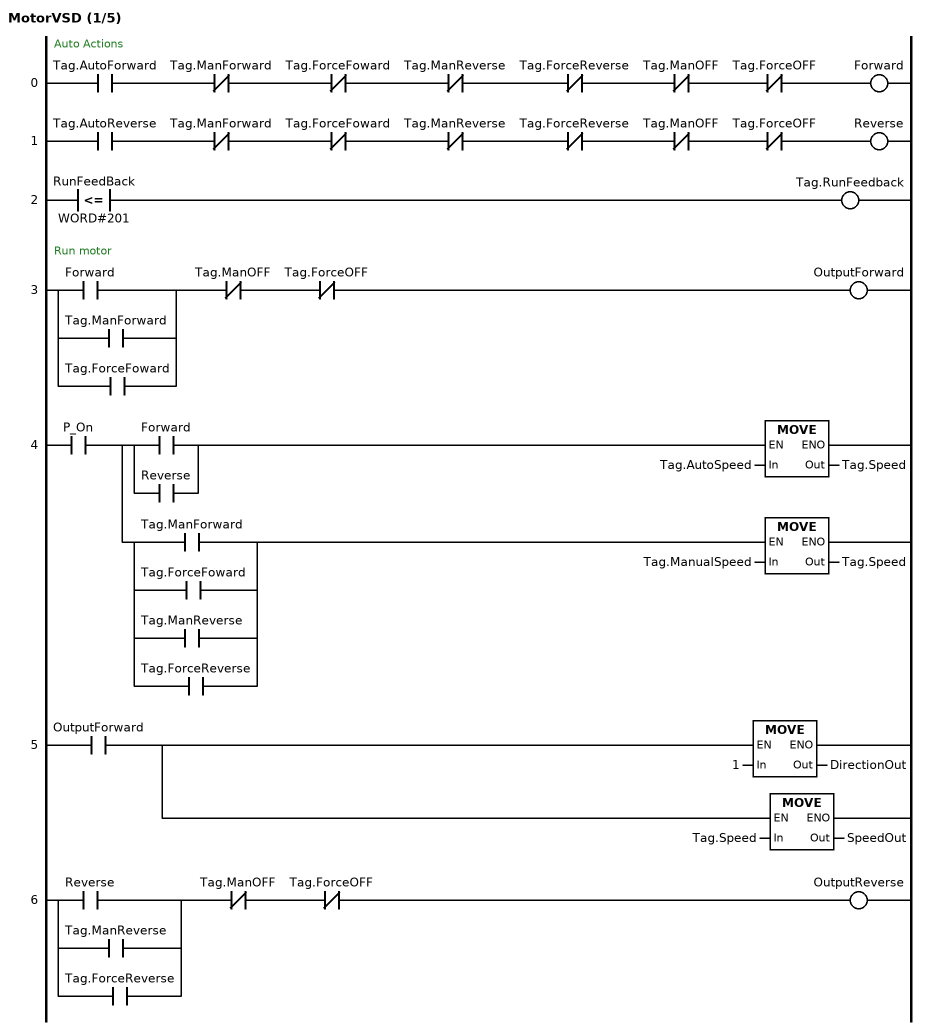
(* Rung 0: Auto Actions *)
Forward := Tag.AutoForward AND NOT Tag.ManForward AND NOT Tag.ForceFoward AND NOT Tag.ManReverse AND NOT Tag.ForceReverse AND NOT Tag.ManOFF AND NOT Tag.ForceOFF;
(* Rung 1 *)
Reverse := Tag.AutoReverse AND NOT Tag.ManForward AND NOT Tag.ForceFoward AND NOT Tag.ManReverse AND NOT Tag.ForceReverse AND NOT Tag.ManOFF AND NOT Tag.ForceOFF;
(* Rung 2 *)
Tag.RunFeedback := RunFeedBack <= WORD#201;
(* Rung 3: Run motor *)
OutputForward := (Forward OR Tag.ManForward OR Tag.ForceFoward) AND NOT Tag.ManOFF AND NOT Tag.ForceOFF;
(* Rung 4 *)
IF P_On AND (Forward OR Reverse) THEN Tag.Speed := Tag.AutoSpeed; END_IF;
IF P_On AND (Tag.ManForward OR Tag.ForceFoward OR Tag.ManReverse OR Tag.ForceReverse) THEN
    Tag.Speed := Tag.ManualSpeed;
END_IF;
(* Rung 5 *)
IF OutputForward THEN
    DirectionOut := 1;
    SpeedOut := Tag.Speed;
END_IF;
(* Rung 6 *)
OutputReverse := (Reverse OR Tag.ManReverse OR Tag.ForceReverse) AND NOT Tag.ManOFF AND NOT Tag.ForceOFF;

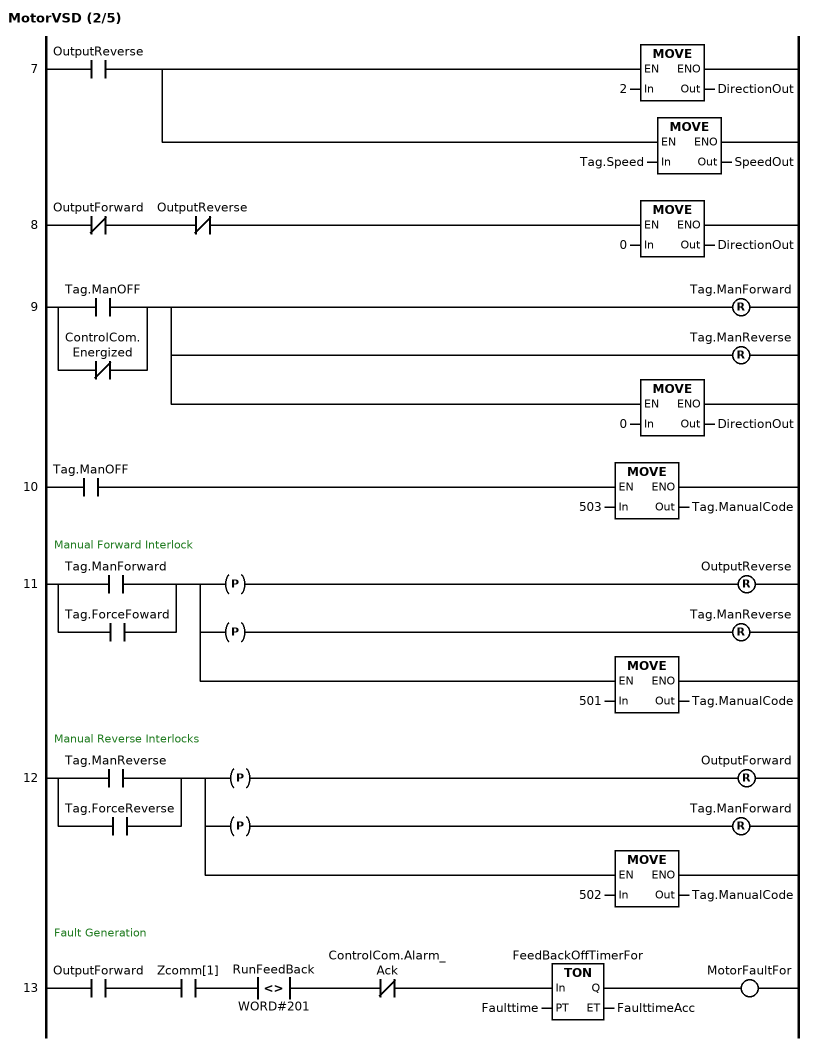
(* Rung 7 *)
IF OutputReverse THEN
    DirectionOut := 2;
    SpeedOut := Tag.Speed;
END_IF;
(* Rung 8 *)
IF NOT OutputForward AND NOT OutputReverse THEN DirectionOut := 0; END_IF;
(* Rung 9 *)
_p1 := Tag.ManOFF OR NOT ControlCom.Energized;
IF _p1 THEN
    Tag.ManForward := FALSE;
    Tag.ManReverse := FALSE;
    DirectionOut := 0;
END_IF;
(* Rung 10 *)
IF Tag.ManOFF THEN Tag.ManualCode := 503; END_IF;
(* Rung 11: Manual Forward Interlock *)
_e2(CLK := Tag.ManForward OR Tag.ForceFoward);
IF _e2.Q THEN OutputReverse := FALSE; END_IF;
_e3(CLK := Tag.ManForward OR Tag.ForceFoward);
_p4 := Tag.ManForward OR Tag.ForceFoward;
IF _e3.Q THEN Tag.ManReverse := FALSE; END_IF;
IF _p4 THEN Tag.ManualCode := 501; END_IF;
(* Rung 12: Manual Reverse Interlocks *)
_e5(CLK := Tag.ManReverse OR Tag.ForceReverse);
IF _e5.Q THEN OutputForward := FALSE; END_IF;
_e6(CLK := Tag.ManReverse OR Tag.ForceReverse);
_p7 := Tag.ManReverse OR Tag.ForceReverse;
IF _e6.Q THEN Tag.ManForward := FALSE; END_IF;
IF _p7 THEN Tag.ManualCode := 502; END_IF;
(* Rung 13: Fault Generation *)
FeedBackOffTimerFor(In := OutputForward AND Zcomm[1] AND (RunFeedBack <> WORD#201) AND NOT ControlCom.Alarm_Ack, PT := Faulttime, ET => FaulttimeAcc);
MotorFaultFor := FeedBackOffTimerFor.Q;

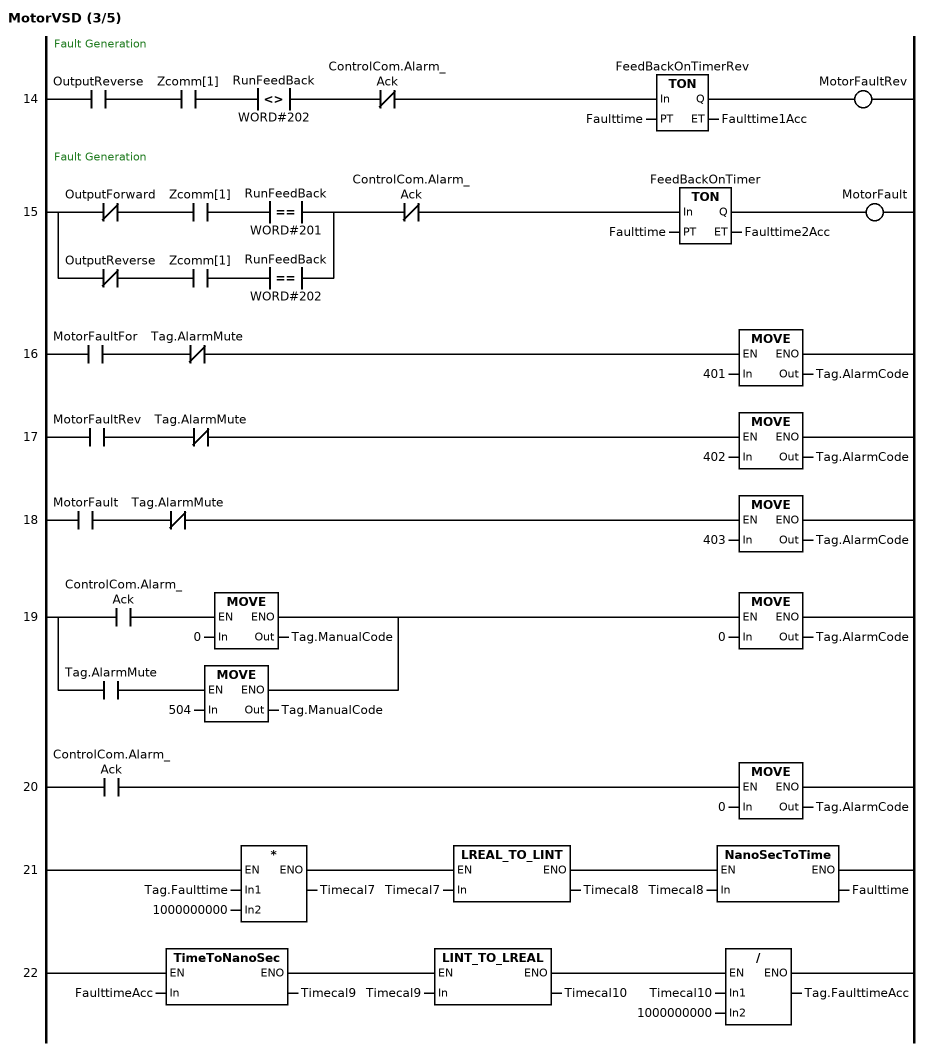
(* Rung 14: Fault Generation *)
FeedBackOnTimerRev(In := OutputReverse AND Zcomm[1] AND (RunFeedBack <> WORD#202) AND NOT ControlCom.Alarm_Ack, PT := Faulttime, ET => Faulttime1Acc);
MotorFaultRev := FeedBackOnTimerRev.Q;
(* Rung 15: Fault Generation *)
FeedBackOnTimer(In := ((NOT OutputForward AND Zcomm[1] AND (RunFeedBack = WORD#201)) OR (NOT OutputReverse AND Zcomm[1] AND (RunFeedBack = WORD#202))) AND NOT ControlCom.Alarm_Ack, PT := Faulttime, ET => Faulttime2Acc);
MotorFault := FeedBackOnTimer.Q;
(* Rung 16 *)
IF MotorFaultFor AND NOT Tag.AlarmMute THEN Tag.AlarmCode := 401; END_IF;
(* Rung 17 *)
IF MotorFaultRev AND NOT Tag.AlarmMute THEN Tag.AlarmCode := 402; END_IF;
(* Rung 18 *)
IF MotorFault AND NOT Tag.AlarmMute THEN Tag.AlarmCode := 403; END_IF;
(* Rung 19 *)
IF ControlCom.Alarm_Ack THEN Tag.ManualCode := 0; END_IF;
_p8 := Tag.AlarmMute;
IF _p8 THEN Tag.ManualCode := 504; END_IF;
IF ControlCom.Alarm_Ack OR _p8 THEN Tag.AlarmCode := 0; END_IF;
(* Rung 20 *)
IF ControlCom.Alarm_Ack THEN Tag.AlarmCode := 0; END_IF;
(* Rung 21 *)
Timecal7 := Tag.Faulttime * 1000000000;
Timecal8 := LREAL_TO_LINT(In := Timecal7);
Faulttime := NanoSecToTime(In := Timecal8);
(* Rung 22 *)
Timecal9 := TimeToNanoSec(In := FaulttimeAcc);
Timecal10 := LINT_TO_LREAL(In := Timecal9);
Tag.FaulttimeAcc := Timecal10 / 1000000000;

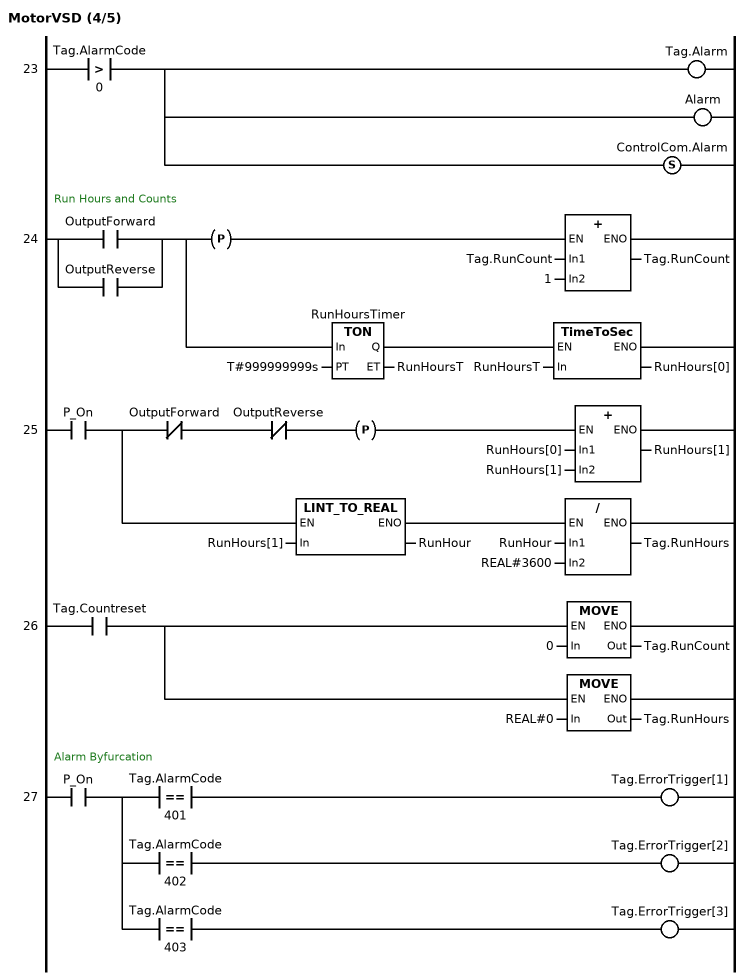
(* Rung 23 *)
_p9 := Tag.AlarmCode > 0;
Tag.Alarm := _p9;
Alarm := _p9;
IF _p9 THEN ControlCom.Alarm := TRUE; END_IF;
(* Rung 24: Run Hours and Counts *)
_e10(CLK := OutputForward OR OutputReverse);
IF _e10.Q THEN Tag.RunCount := Tag.RunCount + 1; END_IF;
RunHoursTimer(In := OutputForward OR OutputReverse, PT := T#999999999s, ET => RunHoursT);
IF RunHoursTimer.Q THEN RunHours[0] := TimeToSec(In := RunHoursT); END_IF;
(* Rung 25 *)
_e11(CLK := P_On AND NOT OutputForward AND NOT OutputReverse);
IF _e11.Q THEN RunHours[1] := RunHours[0] + RunHours[1]; END_IF;
IF P_On THEN
    RunHour := LINT_TO_REAL(In := RunHours[1]);
    Tag.RunHours := RunHour / REAL#3600;
END_IF;
(* Rung 26 *)
_p12 := Tag.Countreset;
IF _p12 THEN
    Tag.RunCount := 0;
    Tag.RunHours := REAL#0;
END_IF;
(* Rung 27: Alarm Byfurcation *)
Tag.ErrorTrigger[1] := P_On AND (Tag.AlarmCode = 401);
Tag.ErrorTrigger[2] := P_On AND (Tag.AlarmCode = 402);
Tag.ErrorTrigger[3] := P_On AND (Tag.AlarmCode = 403);

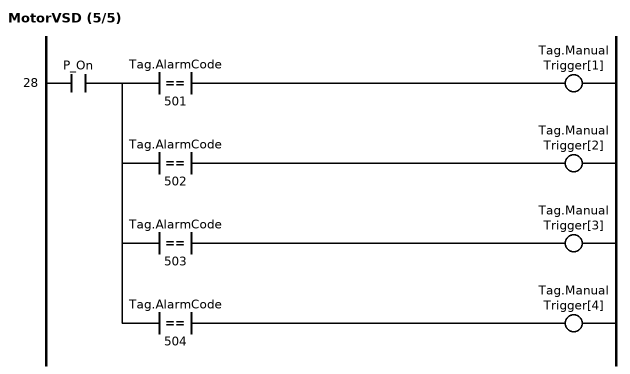
(* Rung 28 *)
Tag.ManualTrigger[1] := P_On AND (Tag.AlarmCode = 501);
Tag.ManualTrigger[2] := P_On AND (Tag.AlarmCode = 502);
Tag.ManualTrigger[3] := P_On AND (Tag.AlarmCode = 503);
Tag.ManualTrigger[4] := P_On AND (Tag.AlarmCode = 504);
END_FUNCTION_BLOCK

FUNCTION_BLOCK MiscOut
VAR
    IN : BOOL;
    Faulttimer : TON;
    FaultTime : TIME;
    FaultTimeAcc : TIME;
    Timecal7 : LREAL;
    Timecal8 : LINT;
    Timecal9 : LINT;
    Timecal10 : LREAL;
END_VAR
VAR_INPUT
    Enable : BOOL;
END_VAR
VAR_OUTPUT
    EnableOut : BOOL;
END_VAR
VAR_IN_OUT
    Tag : MiscOutD;
END_VAR
VAR_INPUT
    Acknowledge : BOOL;
END_VAR
VAR_OUTPUT
    Value : BOOL;
END_VAR
VAR_IN_OUT
    ControlAlarm : BOOL;
END_VAR
VAR
    _p1 : BOOL;
    _p2 : BOOL;
    _p3 : BOOL;
    _e4 : R_TRIG;
    _p5 : BOOL;
    _p6 : BOOL;
END_VAR
(* ladder, written here as Structured Text *)

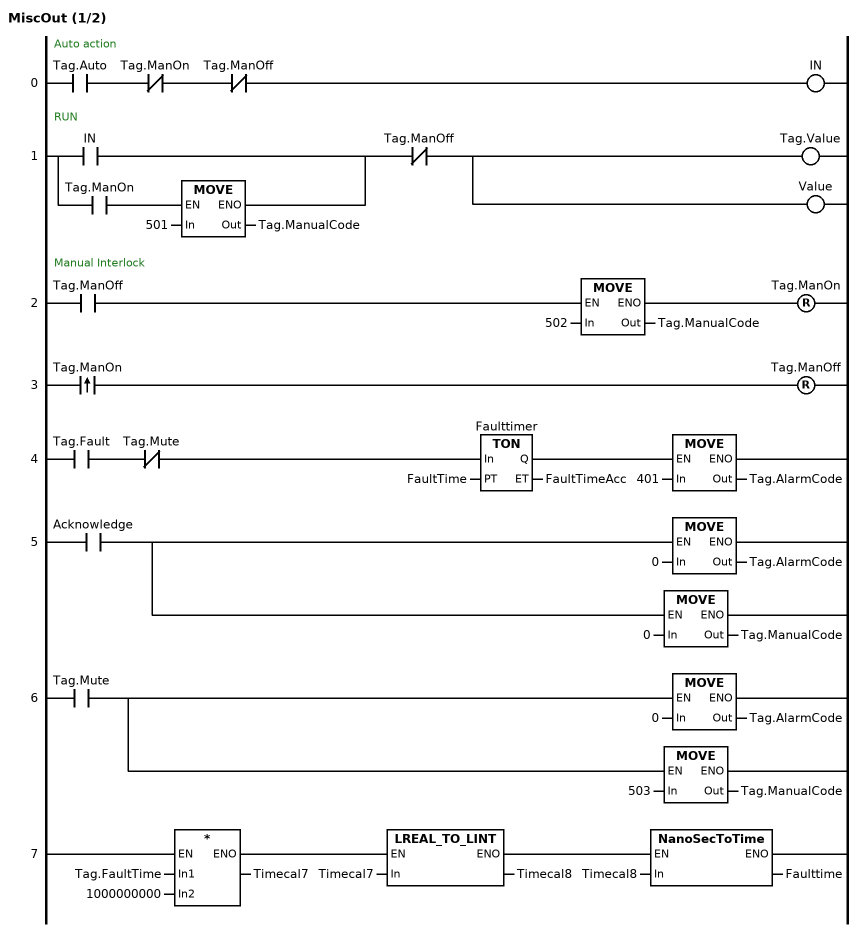
(* Rung 0: Auto action *)
IN := Tag.Auto AND NOT Tag.ManOn AND NOT Tag.ManOff;
(* Rung 1: RUN *)
_p1 := Tag.ManOn;
IF _p1 THEN Tag.ManualCode := 501; END_IF;
_p2 := (IN OR _p1) AND NOT Tag.ManOff;
Tag.Value := _p2;
Value := _p2;
(* Rung 2: Manual Interlock *)
_p3 := Tag.ManOff;
IF _p3 THEN
    Tag.ManualCode := 502;
    Tag.ManOn := FALSE;
END_IF;
(* Rung 3 *)
_e4(CLK := Tag.ManOn);
IF _e4.Q THEN Tag.ManOff := FALSE; END_IF;
(* Rung 4 *)
Faulttimer(In := Tag.Fault AND NOT Tag.Mute, PT := FaultTime, ET => FaultTimeAcc);
IF Faulttimer.Q THEN Tag.AlarmCode := 401; END_IF;
(* Rung 5 *)
IF Acknowledge THEN
    Tag.AlarmCode := 0;
    Tag.ManualCode := 0;
END_IF;
(* Rung 6 *)
_p5 := Tag.Mute;
IF _p5 THEN
    Tag.AlarmCode := 0;
    Tag.ManualCode := 503;
END_IF;
(* Rung 7 *)
Timecal7 := Tag.FaultTime * 1000000000;
Timecal8 := LREAL_TO_LINT(In := Timecal7);
Faulttime := NanoSecToTime(In := Timecal8);

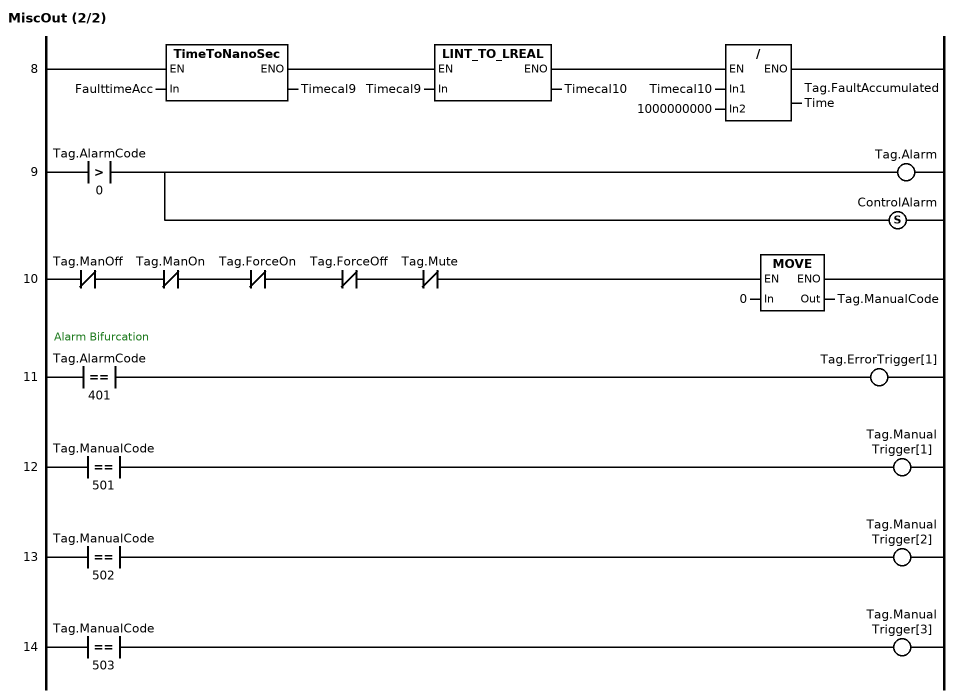
(* Rung 8 *)
Timecal9 := TimeToNanoSec(In := FaulttimeAcc);
Timecal10 := LINT_TO_LREAL(In := Timecal9);
Tag.FaultAccumulatedTime := Timecal10 / 1000000000;
(* Rung 9 *)
_p6 := Tag.AlarmCode > 0;
Tag.Alarm := _p6;
IF _p6 THEN ControlAlarm := TRUE; END_IF;
(* Rung 10 *)
IF NOT Tag.ManOff AND NOT Tag.ManOn AND NOT Tag.ForceOn AND NOT Tag.ForceOff AND NOT Tag.Mute THEN
    Tag.ManualCode := 0;
END_IF;
(* Rung 11: Alarm Bifurcation *)
Tag.ErrorTrigger[1] := Tag.AlarmCode = 401;
(* Rung 12 *)
Tag.ManualTrigger[1] := Tag.ManualCode = 501;
(* Rung 13 *)
Tag.ManualTrigger[2] := Tag.ManualCode = 502;
(* Rung 14 *)
Tag.ManualTrigger[3] := Tag.ManualCode = 503;
END_FUNCTION_BLOCK

FUNCTION_BLOCK StepEngine
VAR
    StepNumChanged : DINT;
    StepTimeAcc : REAL;
    StepTimePre : REAL;
    c : DINT;
    Step1 : DINT;
    i : DINT;
    Currentstep_reset : BOOL;
END_VAR
VAR_INPUT
    EnableIn : BOOL;
END_VAR
VAR_OUTPUT
    EnableOut : BOOL;
END_VAR
VAR_IN_OUT
    Tag : SequenceD;
END_VAR
VAR_INPUT
    ControlCom : System;
END_VAR
VAR
    _p1 : BOOL;
    _p2 : BOOL;
    _p3 : BOOL;
    _p4 : BOOL;
    _p5 : BOOL;
    _p6 : BOOL;
END_VAR
(* ladder, written here as Structured Text *)

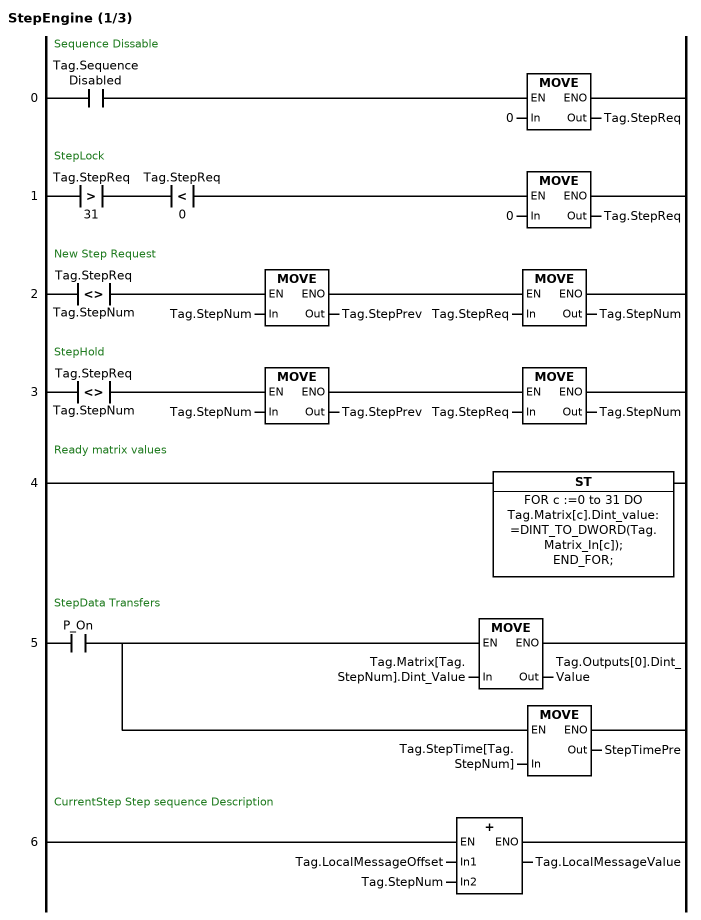
(* Rung 0: Sequence Dissable *)
IF Tag.SequenceDisabled THEN Tag.StepReq := 0; END_IF;
(* Rung 1: StepLock *)
IF (Tag.StepReq > 31) AND (Tag.StepReq < 0) THEN Tag.StepReq := 0; END_IF;
(* Rung 2: New Step Request *)
_p1 := Tag.StepReq <> Tag.StepNum;
IF _p1 THEN
    Tag.StepPrev := Tag.StepNum;
    Tag.StepNum := Tag.StepReq;
END_IF;
(* Rung 3: StepHold *)
_p2 := Tag.StepReq <> Tag.StepNum;
IF _p2 THEN
    Tag.StepPrev := Tag.StepNum;
    Tag.StepNum := Tag.StepReq;
END_IF;
(* Rung 4: Ready matrix values *)
FOR c :=0 to 31 DO
	Tag.Matrix[c].Dint_value:=DINT_TO_DWORD(Tag.Matrix_In[c]);
END_FOR;
(* Rung 5: StepData Transfers *)
IF P_On THEN
    Tag.Outputs[0].Dint_Value := Tag.Matrix[Tag.StepNum].Dint_Value;
    StepTimePre := Tag.StepTime[Tag.StepNum];
END_IF;
(* Rung 6: CurrentStep Step sequence Description *)
Tag.LocalMessageValue := Tag.LocalMessageOffset + Tag.StepNum;

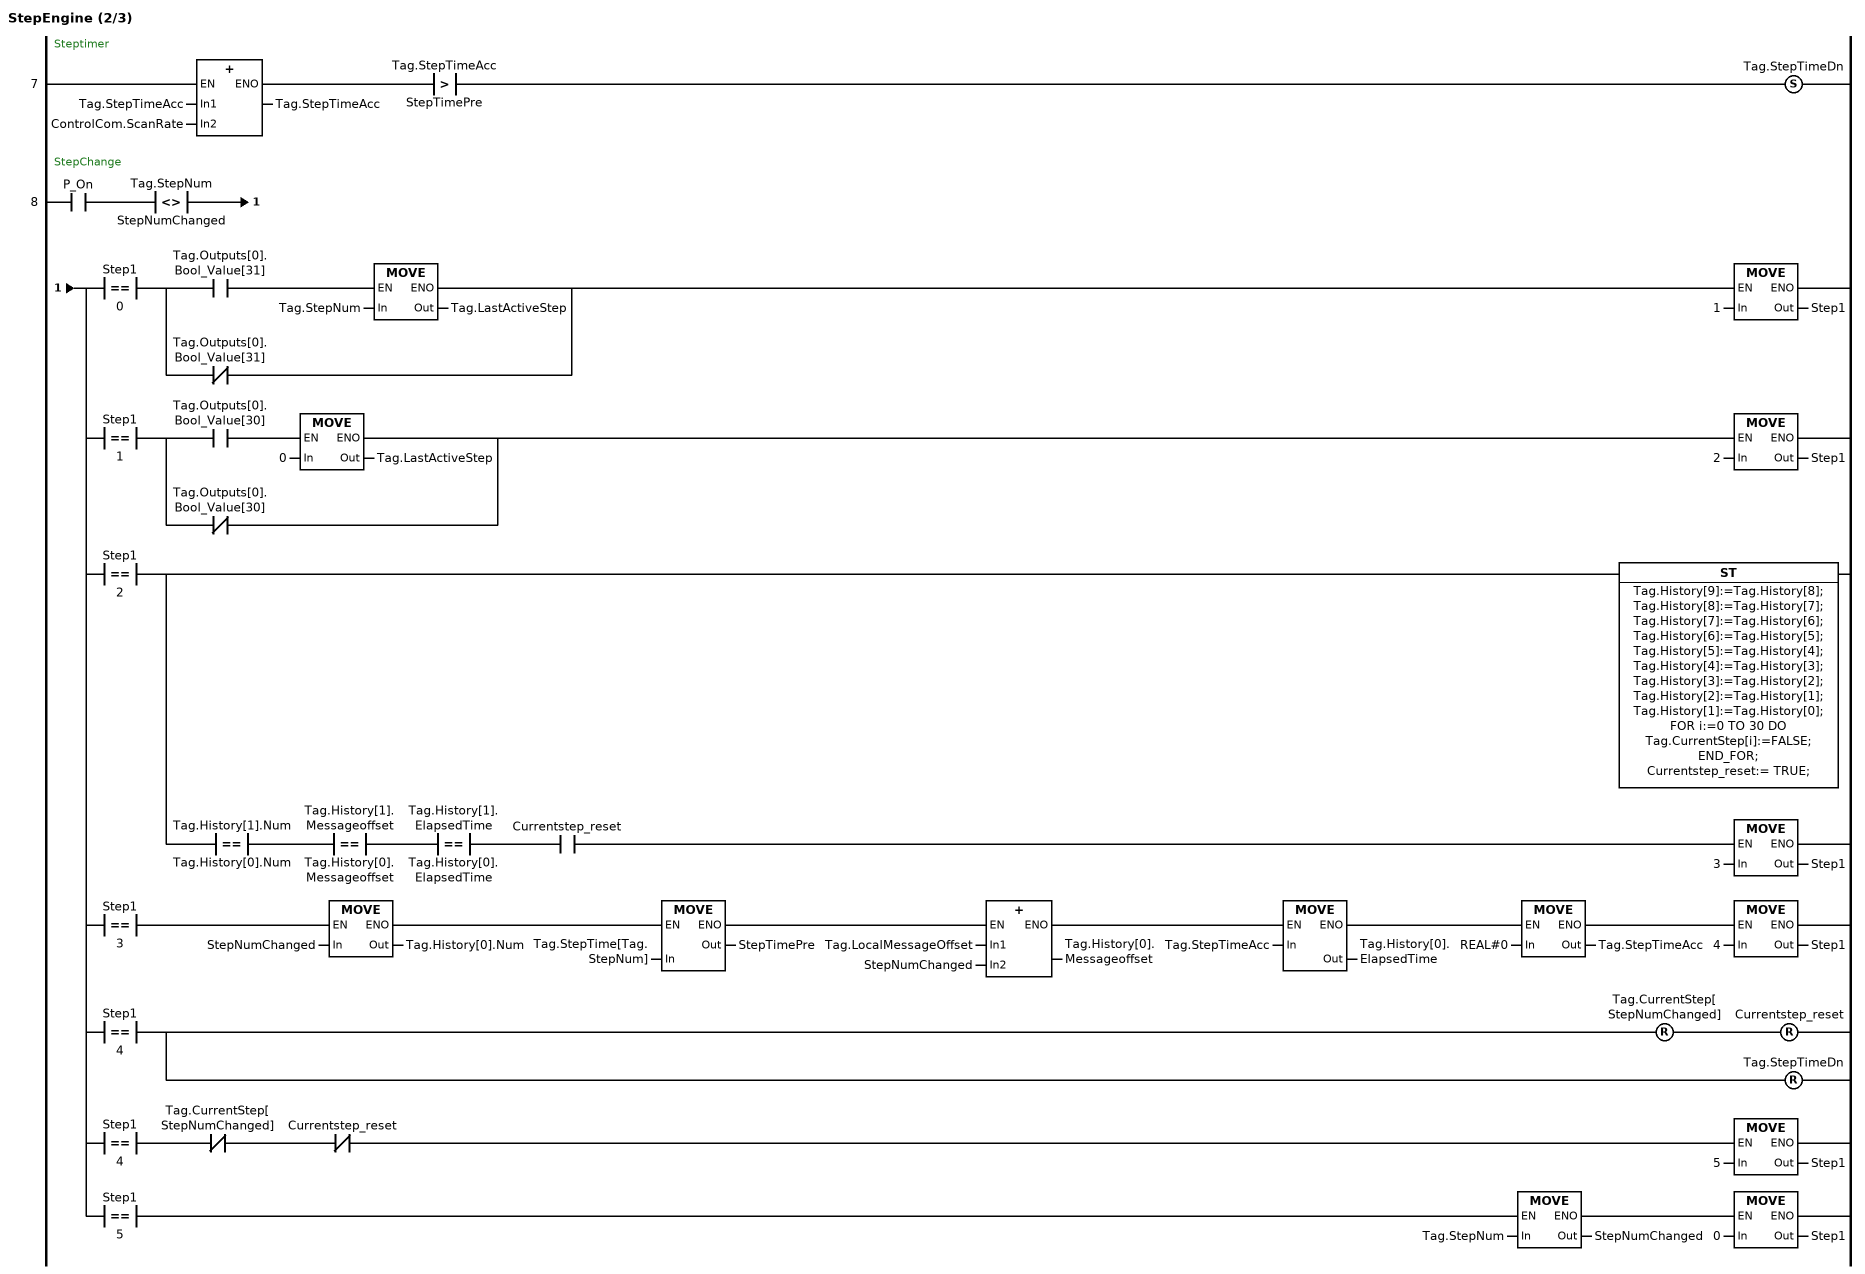
(* Rung 7: Steptimer *)
Tag.StepTimeAcc := Tag.StepTimeAcc + ControlCom.ScanRate;
IF Tag.StepTimeAcc > StepTimePre THEN Tag.StepTimeDn := TRUE; END_IF;
(* Rung 8: StepChange *)
_p3 := P_On AND (Tag.StepNum <> StepNumChanged) AND (Step1 = 0);
_p4 := P_On AND (Tag.StepNum <> StepNumChanged);
_p5 := _p3 AND Tag.Outputs[0].Bool_Value[31];
IF _p5 THEN Tag.LastActiveStep := Tag.StepNum; END_IF;
IF _p5 OR (_p3 AND NOT Tag.Outputs[0].Bool_Value[31]) THEN Step1 := 1; END_IF;
_p6 := _p4 AND (Step1 = 1) AND Tag.Outputs[0].Bool_Value[30];
IF _p6 THEN Tag.LastActiveStep := 0; END_IF;
IF _p6 OR (_p4 AND (Step1 = 1) AND NOT Tag.Outputs[0].Bool_Value[30]) THEN Step1 := 2; END_IF;
IF _p4 AND (Step1 = 2) THEN
    Tag.History[9]:=Tag.History[8];
    Tag.History[8]:=Tag.History[7];
    Tag.History[7]:=Tag.History[6];
    Tag.History[6]:=Tag.History[5];
    Tag.History[5]:=Tag.History[4];
    Tag.History[4]:=Tag.History[3];
    Tag.History[3]:=Tag.History[2];
    Tag.History[2]:=Tag.History[1];
    Tag.History[1]:=Tag.History[0];
    
    FOR i:=0 TO 30 DO
    	Tag.CurrentStep[i]:=FALSE;
    END_FOR;
    
    Currentstep_reset:= TRUE;
END_IF;
IF _p4 AND (Step1 = 2) AND (Tag.History[1].Num = Tag.History[0].Num) AND (Tag.History[1].Messageoffset = Tag.History[0].Messageoffset) AND (Tag.History[1].ElapsedTime = Tag.History[0].ElapsedTime) AND Currentstep_reset THEN
    Step1 := 3;
END_IF;
IF _p4 AND (Step1 = 3) THEN
    Tag.History[0].Num := StepNumChanged;
    StepTimePre := Tag.StepTime[Tag.StepNum];
    Tag.History[0].Messageoffset := Tag.LocalMessageOffset + StepNumChanged;
    Tag.History[0].ElapsedTime := Tag.StepTimeAcc;
    Tag.StepTimeAcc := REAL#0;
    Step1 := 4;
END_IF;
IF _p4 AND (Step1 = 4) THEN
    Tag.CurrentStep[StepNumChanged] := FALSE;
    Currentstep_reset := FALSE;
    Tag.StepTimeDn := FALSE;
END_IF;
IF _p4 AND (Step1 = 4) AND NOT Tag.CurrentStep[StepNumChanged] AND NOT Currentstep_reset THEN
    Step1 := 5;
END_IF;
IF _p4 AND (Step1 = 5) THEN
    StepNumChanged := Tag.StepNum;
    Step1 := 0;
END_IF;

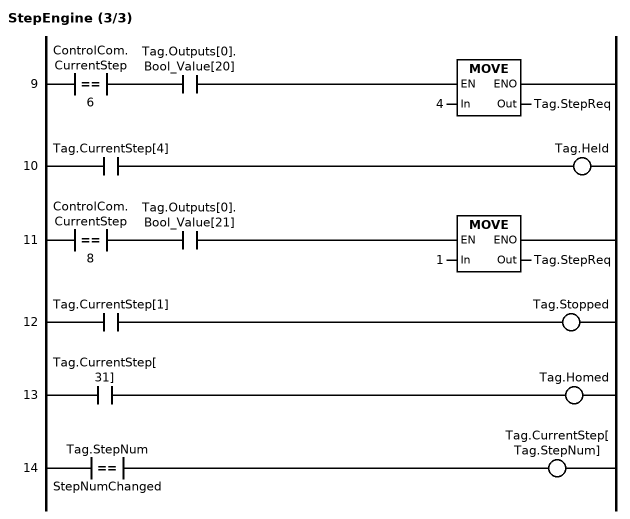
(* Rung 9 *)
IF (ControlCom.CurrentStep = 6) AND Tag.Outputs[0].Bool_Value[20] THEN Tag.StepReq := 4; END_IF;
(* Rung 10 *)
Tag.Held := Tag.CurrentStep[4];
(* Rung 11 *)
IF (ControlCom.CurrentStep = 8) AND Tag.Outputs[0].Bool_Value[21] THEN Tag.StepReq := 1; END_IF;
(* Rung 12 *)
Tag.Stopped := Tag.CurrentStep[1];
(* Rung 13 *)
Tag.Homed := Tag.CurrentStep[31];
(* Rung 14 *)
Tag.CurrentStep[Tag.StepNum] := Tag.StepNum = StepNumChanged;
END_FUNCTION_BLOCK

FUNCTION_BLOCK Vision
VAR
    TriggerUp : BOOL;
    TriggerOld : BOOL;
END_VAR
VAR_INPUT
    EnableIn : BOOL;
END_VAR
VAR_OUTPUT
    EnableOut : BOOL;
END_VAR
VAR_IN_OUT
    ScannerI : ScannerD;
    ControlComm : System;
END_VAR
VAR_INPUT
    Vision_In : Vis_In;
END_VAR
VAR_OUTPUT
    Vision_Out : Vis_out;
    Alarm : BOOL;
END_VAR
VAR
    _e1 : R_TRIG;
    _p2 : BOOL;
END_VAR
(* ladder, written here as Structured Text *)

